	(*śmieci*)
	tonExecute															: TON;		
	tonNotExecute														: TON;	
	tonDelayAfterStart6s              									: TON;
	tonReadedCardFirstDelayBottleTransfer								: TON;
	tonReadedCardSecondDelayBottleTransfer								: TON;
	tonFourthFormatSensor												: TON;
	tonFourthFormatSensor2												: TON;	
	tonThirdFormsSensor													: TON;
	tonWaitUntilSecondFormPresent										: TON;
	tonLongDelayFirstDraging											: TON;
	tonLongDelayFirstDragingLidFeeder									: TON;	
	tonLongDelayFirstDragingLidSealer									: TON;	
	tonWeightBeforeGateDispSensor										: TON;
	tonBeforeGateSensorDelay											: TON;
	tonTransporterStopping												: TON;
	TimerCycleReseting													: TON;
	tonAfterScreweEmpty													: TON;
	tonCapCorrectCheckAfterScrewerFormSensor							: TON;
	fbbCapCorrectCheckAfterScrewerFormSensor							: FB_InputFilter_v2;
	tonDelayAfterReset													: TON;
	tonCycleLabelMachineFullSensor										: TON;
	tonCycleBadBottleConveyorFullSensor									: TON;
	tonCycleBadBottleConveyorFullSensor2								: TON;
	tofBadBottleConveyorStart											: TOF;
	tofbFormTransportersDispencerSlow									: TOF;
	tonbFormTransportersDispencerResetSpeed								: TON;
	tonQueBeforeScrewers												:TON;
	tonQueAfterScrewers													:TON;
	tonTimer4thFormBeforeCapSorter										:TON;
	tonQueAfterPlatin													:TON;
	tonQueBeforeDispencers												:TON;
	tonDelayedStartAfterDisp											:TON;
	
	i																	: UINT;
	nCheckCountR4														: UINT;
	iFormatOnWeightCounter												: UINT;
	cpc																	: INT;
	nccc																: INT;
	iBottleTransferCase													: INT;
	nCheckCountR1														: INT;
	iii																	: INT;
	iDispDragCase														: INT;
	iWeightCase															: INT;
	iScrewerDragCase													: INT;
	nw																	: INT;
	nw3																	: INT;
	nw2																	: INT;
	nw4																	: INT;
	nw5																	: INT;
	nw6																	: INT;
	nCounterFormsToLoad													: INT;
	nCounterForms														: INT;
	z																	: INT;
	iRobotPickCase														: INT;
	y																	: INT;
	nCounterCase7														: INT;
	nCounterCase8														: INT;
	nCounterCase10														: INT;
	nCounterCase14														: INT;
	nCounterCase11														: INT;
	nCounterCase12														: INT;
	cch																	: INT;
	cchc																: INT;	
	jw1																	: INT;
	jw2																	: INT;
	iw3																	: INT;
	jw3																	: INT;
	iw4																	: INT;
	jw4																	: INT;
	iw5																	: INT;
	jw5																	: INT;
	iw6																	: INT;
	jw6																	: INT;
	ic1																	: INT;
	iCOunterTest10														: INT;
	iWeightOnFormCase													: INT;
	nCountTest2															: INT;
	nCountTest3															: INT;
	iGateDispCase														: INT;
	counterchecked														: INT;
	nCounterCase9														: INT;
	nCounterCase13														: INT;
	nCounterCase15														: INT;
	ibRobotPackageState1NOK												: INT;
	iBeforeDispencerCounter												: INT;
	bRobotCycleRFIDReadedOne											: BOOL;
	bRobotCycleRFIDReadedTwo											: BOOL;
	bBadBottleConveyorStartTrigger										: BOOL;
	bBadBottleConveyorStartTriggerDelay									: BOOL;	
	bRobotGateStayOpen													: BOOL;
	bRobotPackageState1OK												: BOOL;
	bRobotPackageState1NOK												: BOOL;
	bRobotPackageState2OK												: BOOL;
	bRobotPackageState2NOK												: BOOL;
	bRobotPackageState1Rotate											: BOOL;
	bRobotPackageState2Rotate											: BOOL;
	iChangeModeStep: INT;
	bCatchersReady2														: BOOL;
	bDispencer2CatchedOrNoBottle										: BOOL;
	bDispencer1CatchedOrNoBottle										: BOOL;
	bDispencer3CatchedOrNoBottle										: BOOL;
	bDispencer4CatchedOrNoBottle										: BOOL;
	bCounterDisabled													: BOOL;
	bRobotPackageState1Empty											: BOOL;
	bRobotPackageState2Empty											: BOOL;
	//ctdCounterFormOnRobot												: CTD;
	iResetAfterErrorOrEstop: INT;
	iBeforeDispencer2PhaseCounter: INT;
	bBottleFeederHommed: BOOL;
	iFormatOnWeight2PhaseCounter: UINT;
	tonCheckFourthFormNotPresent: TON;
	tonFourthFormat2PhaseSensor: TON;
	tonCheckFormSensorBetweenDispencer: TON;
	ftfbIbWeightFirstForm2PhaseSensor: F_TRIG;
	iPhaseChangingStep: INT;
	tonPhaseChangingCase110Delay: TON;
	tonPhaseChangingCase200Delay: TON;	
	tonPhaseChangingCase210Delay: TON;
	iTestDrag: INT;
	brtLongDelayFirstDraging: BOOL;
	bFirstDragingLidFeederAfterRestart1: BOOL;	
	bFirstDragingLidFeederAfterRestart2: BOOL;	
	bFirstDragingLidSealerAfterRestart1: BOOL;	
	bFirstDragingLidSealerAfterRestart2: BOOL;		
	tonSecondForm2PhaseSensor: TON;
	bPhaseChangingGatePermission: BOOL;
	brtLongDelayFirstDragingDone: BOOL;
	brtLongDelayFirstDragingLidFeederDone: BOOL;	
	bDelayAfterStartFullRegister: BOOL;
	tonSecondForm2PhaseSensorRepair: TON;
	tonGripperScrewerDragMiddleSensor: TON;
	tonDispencersDragLeftMiddleSensor: TON;
	tonDispencersDragRightMiddleSensor: TON;
	tonDelayAfterBottleFeederDoorOpen: TON;
	tonCheckFormBeforeDispencersGate: TON;
	fbIbFourthFormCheckFormSensor: FB_InputFilter_v2;
	fbIbTwoPhasesFormSensorBetweenDispencers: FB_InputFilter_v2;
	fbIbSecondFormCheckFormSensor: FB_InputFilter_v2;
	tofbDosingTwoPhases:TOF;
	tonNotLongDelayAfterStart: TON;
	nVarModuloSimulation: INT;
	tonNotReadedCardFirstDelayBottleTransfer: TON;
	tonNotReadedCardSecondDelayBottleTransfer: TON;
	fbIbBottleTransferFormAfterSensor: FB_InputFilter_v2;
	rttonNotReadedCardFirstDelayBottleTransfer: R_TRIG;
	rttonNotReadedCardSecondDelayBottleTransfer: R_TRIG;
	iCounterRepairNotReadedFirst: INT;
	iCounterRepairNotReadedSecond: INT;
	rtbRobotPackageState1NOK: R_TRIG;
	rtbRobotPackageState2NOK: R_TRIG;
	ibRobotPackageState2NOK: INT;
	fbIbGripperScrewersThirdFormCheckFormSensor:FB_InputFilter;
	fbIbGripperScrewersBeforeThirdFormCheckFormSensor:FB_InputFilter;
	tofFormsDragingPneumaticStationDraged	:	TOF;
	toffbDispencersDragLeftStationbCycleDone: TOF;
	tonWeight14CycleDoneAndCase: TON;
	tonWeight56CycleDoneAndCase: TON;	
	iFormTransportersScrewerResetSpeedPulse: INT;

	
	(*CapSorter*)
	tonCapSorterDragMiddleSensor			:TON;
	tonIbCapSorterAfterFormSensor			:TON;
	tonIbCapSorterAfterFormSensor3			:TON;	
	brtCapSorterLongDelayFirstDraging		:BOOL;
	bCapSorterDragIfNot4PucksAnd5s			:BOOL;	
	tonCapSorterDragIfNot4PucksAnd5s		:TON;
	tonCapSorterFourthFormatSensorAnRegister:TON;
	tonIbCapSorterFirstFormCheckFormSensor	:TON;
	tonCapSorterFourthFormatSensor			:TON;
	tonCapSorterFourthFormatSensorStarting	:TON;	
	tonbFormTransportersAfterCapSorterCmdStart:TON;
	rttonCapSorterFourthFormatSensorCounter	:R_TRIG;
	tonCapSorterDragFormCounter4			:TON;
	tonCapSorterDragFormCounter4b			:TON;	
	itonCapSorterDragFormCounter4			:INT;
	itonCapSorterDragFormCounter4b			:INT;
	tonStoppingCapSorter					:TON;
	tonCapSorterDelay						:TON;
	tonCapSorterDelay2						:TON;
	iCapSorterCase							:INT;
	bDelayAfterStartCapSorterFullRegister	:BOOL;
	(*inne*)
	//Vasyl 30.05 
	tonPucksInserterPushTableOff			:TON;

	(*Szalaban przed waga*)
	iWeightGateBeforeCASE					: INT;													
	
	(*Zatrzymywanie transportera*)
	tonCapSorterCycleTime					: TON;
	fttonCapSorterCycleTime					: F_TRIG;
	AtCapSorterCycleTime					: ARRAY [1..100] OF TIME;
	bCapSorterCycleTest						: BOOL ;
	tonCapSorterPackageState1bCapSorterPutted: TON;
	tCapSorterCycleTestTime					: TIME;
	
	(*Wbijak butelek*)
	bBottlePusherBottleBeforeSensor			: BOOL;
	tonBottlePusherBottleBeforeSensor		: TON;
	
	
	(*AutoStart ADS*)
	tonBottleSorterAutoStart 				: TON;
	tonCapSorterAutoStart					: TON;
	iBottleSorterAutoStart 					: INT;	
	iCapSorterAutoStart						: INT;
	bCapSorterBottleSorterAutoStart 		: BOOL;	
	tonbCapSorterBottleSorterAutoStart 		: TON;
	
	(*Dodatkowe sprawdzanie butelki*)

	rtIbCapCorrectCheckFormSensor			: R_TRIG;
	
	(*Inne*)
	
	iAbortingTest: INT;
	iChooseRecipe: INT;

	toniWeight14GateBeforeCASE: TON;
	toniWeight14GateBeforeCASE2: TON;
	fbIbWeight14Gate4FormBeforeSensor: FB_InputFilter_v2;
	tonbGateBeforeWeight14Run: TON;
	toniWeight56GateBeforeCASE: TON;
	toniWeight56GateBeforeCASE2: TON;
	fbIbWeight56Gate6FormBeforeSensor: FB_InputFilter_v2;
	tonbGateBeforeWeight56Run: TON;
	
	ics: INT;
	ttonCapSorterCycleTimeET: TIME;
	bCapSorterError: BOOL;
	tonbCapSorterError: TON;
	tonbCapSorterOrCapSorterDragError: TON;	
	fbDrand: DRAND;
	diRandom :DINT;
	iTestResetCommandsStopped: INT;
	tonCapSorterHomingAndDone: TON;
	tonBottleSorterHomingAndDone: TON;
	irtResetAfterStart: INT;
	ibDelayAfterStartCapSorterFullRegister: INT;
	toniHomingCase20: TON;
	iTestiHomingCase: INT;

	bStopping1Weight: BOOL;
	bStoppingWeight1: BOOL;
	bStoppingWeight2: BOOL;
	bStoppingWeight3: BOOL;
	bStoppingWeight4: BOOL;
	tonStoppingBottleTransfer1: TON;
	
	tonbFirstCycle: TON;
	iTestW: INT;
	
	(*Wydmuch przed zakręcarkami*)
	fbIbBlowBeforeGripperScrewerSensor	:	FB_InputFilter_v2;
	fbIbBlowBeforeGripperScrewerSensor2	:	FB_InputFilter_v2;
	
	(*Licz form. przed doz*)
	rtIbFourthFormCheckFormSensor:	R_TRIG;
	tonIbFourthFormCheckFormSensor: TON;
	tonFormsDragingFormCounter4	: TON;
	tonFormsDragingFormCounter4b: TON;	
	itonFormsDragingFormCounter4: INT;	
	itonFormsDragingFormCounter4b: INT;
	
	(*Szlaban przed zakrecarkami*)
	fbIbGateBeforeGripperScrewerSensor						: FB_InputFilter;
	fb2IbGateBeforeGripperScrewerSensor						: FB_InputFilter;	
	ftfbIbGateBeforeGripperScrewerSensor					: F_TRIG;
	bGateBeforeGripperScrewer								: BOOL;
	tonbGateBeforeGripperScrewer							: TON;
	
	(*Lid Feeder Drag*)
	iLidFeederDragCase										: INT;	
	tofbLidFeederDragingStationPrepareRun					: TOF;
	tonLidFeederFirstFormSensorBeforeDrag					:TON;
	iLidFeederDragStoppingCount								: INT;
	bLidFeederDragDelayAfterStartFullRegister				: BOOL;	
	tonLidFeederDragSecondFormSensor						: TON;
	fbIbLidFeederAfterSensor								: FB_InputFilter_v2;
	fbIbLidFeederAfterSensorLonger							: FB_InputFilter_v2;
	tonAfterLidFeederEmpty									: TON;
	tonLidFeederThirdFormsSensor							: TON;
	fbIbLidFeederThirdFormCheckFormSensor					: FB_InputFilter_v2;
	bLidFeederReady											: BOOL;
	fb2IbLidFeederThirdFormSensor							: FB_InputFilter_v2;
	tonStartLidFeederDelay									: TON;
	iLidFeederCase											: INT;
	tonfbLidFeederDragStationNotbCycleDone					: TON;		
	(*Lid Putted Check*)
	fbIbLidPuttedCheck1Sensor								: FB_InputFilter_v2;
	fbIbLidPuttedCheck2Sensor								: FB_InputFilter_v2;
	
	
	(*Lid Sealer Drag*)
	iLidSealerDragCase										: INT;
	tofbLidSealerDragingStationPrepareRun					: TOF;
	iLidSealerDragStoppingCount								: INT;
	bLidSealerDragDelayAfterStartFullRegister				: BOOL;	
	tonLidSealerDragSecondFormSensor						: TON;
	fbIbLidSealerAfterSensor								: FB_InputFilter_v2;
	fbIbLidSealerAfterSensor2								: FB_InputFilter_v2;
	tonLidSealerThirdFormsSensor							: TON;
	tonLidSealerFirstFormsSensor								: TON;
	fbIbLidSealerThirdFormCheckFormSensor					: FB_InputFilter_v2;
	bLidSealerReady											: BOOL;
	fb2IbLidSealerSecondFormSensor							: FB_InputFilter_v2;
	fbNotIbLidSealerSecondFormSensor							: FB_InputFilter_v2;	
	tonStartLidSealerDelay									: TON;
	iLidSealerCase											: INT;	
	tonbFormTransportersScrewerCmdStart						: TON;
	tonfbLidSealerDragStationNotbCycleDone					: TON;		
	rttonLidSealerSecondFormatSensorCounter					: R_TRIG;
	tonLidSealerSecondFormatSensor							: TON;
	tonLidSelaerDragIfNot2PucksAnd5s						: TON;
	bLidSelaerDragIfNot2PucksAnd5s							: BOOL;
	(*Transfer na wagę*)
	udiBottleTransferWeightIntervalCount: UDINT;
	bBottleTransferDoWeight: BOOL;
	
	(*Inne*)
	iGateBeforeGripperScrewerCase: INT;
	toniGateBeforeGripperScrewerCase1: TON;
	tonBadBottleConveyorStop: Ton;
	
	
	toWeightRealeseByLidFeeder: TON;

	tonbFormTransportersScrewerStop: TON;
	tofFormTransportersScrewerSlowSpeed: TOF;
	iFirstDragingLidFeederAfterRestart2Count: INT;
	iFirstDragingLidSealerAfterRestart2Count: INT;	
	tonP13_BottleTransferfbBottleTransfereRunningStateeRejecting: TON;
	nUnderCorrectCapPackageStateLastnCardNumber: ULINT;
	nCapCorrectCheckCameraNOK: INT;
	rtP11_CapCorrectCheckfbCapCorrectCheckCamerabCycleDone: R_TRIG;
	nCapCorrectCheckCameraOK: INT;
	tonDragAE1: TON;
	
	(*Spowalniacz*)
	tonCapPuttedFormsCheck						:	TON;
	tonThirdFormCheckFormSensor					:	TON;
	
	(*SignalFormCounting*)
	fbIbCapSorterGateScrewerSensor: FB_InputFilter_v2;
	fbIbCapSorterGateWeightSensor: FB_InputFilter_v2;
	fbIbCapCorrectCheckFormSensor: FB_InputFilter_v2;

	(*PucksInserter*)
	bPucksInserterHommed: BOOL;

	(*inne*)
	iSetNumbersOfFormsBetweenWeightAndScrewers: INT;
	tofCapCorrectCheckAfterScrewerFormSensor: TOF;

	itonWeightPackageState1BnNoCardNumber: INT;
	itonWeightPackageState2BnNoCardNumber: INT;
	itonWeightPackageState3BnNoCardNumber: INT;
	itonWeightPackageState4BnNoCardNumber: INT;
	tonBreakpoint: TON;
	bBreakpoint: BOOL;
	tontonDelayAfterStart: TON;
	tonDelayForGatePI: TON;
	tonIbPucksInserterFormGateBeforeSensor: TON;

	(*ROPP*)
	fbIbROPPThirdFormSensor					:FB_InputFilter_v2; 
	rtfbIbROPPThirdFormSensor				:R_TRIG;
	rtfbIbROPPThirdFormSensor2				:R_TRIG;	
	ftfbIbROPPThirdFormSensor				:F_TRIG;
	tonROPPThirdFormSensor					:TON;
	tonROPPThirdFormSensor2					:TON;
	tonROPPAfterFormSensor					:TON;
	fbIbROPPAfterFormSensor 				:FB_InputFilter_v2; 
	fbIbROPPAfterFormSensor2 				:FB_InputFilter_v2; 
	fbIbROPPAfter3FormSensor 				:FB_InputFilter_v2; 
	ftIbROPPAfterFormSensor 				:F_TRIG; 
	iROPPAfterFormCounter					:INT;
	iROPPBeforeFormCounter					:INT;
	iTestRop1:INT;
	fbIbROPPSevenFormSensor					:FB_InputFilter_v2; 
	fbIbROPPSevenFormSensor2				:FB_InputFilter_v2; 
	rtfbIbROPPSevenFormSensor2				:R_TRIG;
	ftfbIbROPPSevenFormSensor2				:F_TRIG;
	ftbReadedCardBeforeROPP					:F_TRIG;
	tonbReadedCardBeforeROPP				:TON;
	fbbReadedCardAfterROPP					:FB_InputFilter_v2; 
	rtfbbReadedCardAfterROPP				:R_TRIG;
	ftfbbReadedCardAfterROPP				:F_TRIG;	
	rpc,rpc1,rcc,rcc1						:INT;
	bROPPReady								:BOOL;
	bROPPDelayAfterStartFullRegister		:BOOL;
	tonROPPStartCappingDelay				:TON;
	tofbROPPCappingRunEngine				:TOF;
	iROPPCappingCase						:INT;
	rtiROPPAfterFormCounter0				:R_TRIG;
	bDragTest								:BOOL;
	fbROPPIbCapSorterBeforeFourthFormCheckFormSensor:FB_InputFilter_v2; 
	iTestBot :INT;
	bTestBot:BOOL;
	BtESTbOT1:BOOL;
	iFormBeforeScrewers:INT;
	iFormBeforeROPP:INT;
	//bBlowBeforeGripperScrewer:BOOL;
	//tonbBlowBeforeGripperScrewer:TON;
	//tonQbBlowBeforeGripperScrewer:TON;
	tonIbROPPBeforeSevenFormSensor:TON;
	tpfbIbBlowBeforeGripperScrewerSensor:TP;
	iCaseSingleRealeseIfNoCapFromScrewersPulse:INT;
	tonSingleRealeseIfNoCapFromScrewers1:TON;
	tonSingleRealeseIfNoCapFromScrewers2:TON;	
	bSingleRealeseIfNoCapFromScrewersDragBlock: BOOL;
	rtSingleRealeseIfNoCapFromScrewers1:R_TRIG;
	rtSingleRealeseIfNoCapFromScrewers2:R_TRIG;
	tonBlowBeforeGripperScrewerSensor: TON;
	fbIbPucksInserterFormGateAfterSensor :FB_InputFilter_v2;
	fbIbPucksInserterPushTablesSensor :FB_InputFilter_v2;
	tofIbCapCorrectCheckFormSensor:TOF;
	bCapCorrectCheckBottleSensorLast:BOOL;
	iCapCorrectCheckBottleSensorLast:INT;
	bCapSorterDragIfNot4PucksAnd5sRepair:BOOL;
	fbTransporterQueues: FB_InputFilter_V2;
	fbIbDispencerAfterCheckFormSensor: FB_InputFilter_v2;
	fbIbDispencer12NoColisionWhenDosingSensor: FB_InputFilter_v2;
	fbIbDispencer34NoColisionWhenDosingSensor: FB_InputFilter_v2;	
	fbIbCapSorterFourthFormCheckFormSensor: FB_InputFilter_v2;
	rttofIbCapCorrectCheckFormSensor: R_TRIG;
	ibFormsDragingRightRun:INT;
	ibFormsDragingLeftRun:INT;	
	ftbFormsDragingRightRun:F_TRIG;
	ftbFormsDragingLeftRun:F_TRIG;
	rtbFormsDragingLeftRun	:R_trig;
	rtbFormsDragingRightRun	:R_trig;
	
	(*Szlaban na trans odbviorczym*)
	fbIbExitConveyorGateAfterSensor		:FB_InputFilter_v2;
	fbIbExitConveyorGateAfterSensor2	:FB_InputFilter_v2;	
	fbIbExitConveyorGateAfterSensor3	:FB_InputFilter_v2;	
	tonbExitConveyorGateRun				:TON;
	bExitConveyorGateRunTemp			:BOOL;
	(*Koniec Szlaban na trans odbviorczym*)
	bSafetyTest							:BOOL;
	
	lrGripperScrewerStoperPosition		:LREAL;
	tpGripperScrewerStoperTimerOn		:TP;	// timer do generowania impulsu
	fbGripperScrewerStoperSensorDelay	:FB_InputFilter;	// filtr do generowania sygnału 
	tofQbGripperScrewerStoperActuator	:TOF;	
	rtQbGripperScrewerStoperActuator	:R_TRIG;
	fbQbGripperScrewerGateBeforeActuator:FB_InputFilter_v2;	
	rtfbQbGripperScrewerGateBeforeActuator:R_TRIG;	
	bGripperScrewerStoper2ReadyToDrag 	:BOOL;
	tonQbGripperScrewerGateBeforeActuator:TON;
	itestdpvs			:INT;
	itestdpvs2			:INT;
	itestdpvs3			:INT;	
	bEXPACK	:BOOL:=FALSE;
	tofWeight6FormSensor	:TOF;
	tofbacktodrag			:TOF;
	tofQueAfterPlatinForDisp	:TOf;
	tonQueBeforePlatins	:TON;
	bGripperScrewerAcceleratorActuatorTemp: BOOL;
	tonDelayLid1Putting	:TON;
	tonDelayLid2Putting	:TON;
	
	
	//P13_BottleTransferAfterDrag
	tonBottleTransferAfterDrag	: TON;
	fbIbBottleTransferAfterDragAfterSensor : FB_InputFilter_v2;
	fbIbBottleTransferAfterDragSecondFormSensor	 : FB_InputFilter_v2;
	rtfbIbBottleTransferAfterDragSecondFormSensor : R_TRIG;
	rtfbIbBottleTransferAfterDragSecondFormSensorCounter : INT;
	tonrtfbIbBottleTransferAfterDragSecondFormSensorCounter: TON;
	// Konie cP13_BottleTransferAfterDrag
	
	(*Wick Feeder*)
	iWickFeederDragCase										: INT;	
	tofbWickFeederDragingStationPrepareRun					: TOF;
	tonWickFeederFirstFormSensorBeforeDrag					:TON;
	iWickFeederDragStoppingCount							: INT;
	bWickFeederDragDelayAfterStartFullRegister				: BOOL;	
	tonWickFeederDragSecondFormSensor						: TON;
	fbIbWickFeederAfterSensor								: FB_InputFilter_v2;
	fbIbWickFeederAfterSensorLonger							: FB_InputFilter_v2;
	tonAfterWickFeederEmpty									: TON;
	tonWickFeederThirdFormsSensor							: TON;
	fbIbWickFeederThirdFormCheckFormSensor					: FB_InputFilter_v2;
	bWickFeederReady										: BOOL;
	fb2IbWickFeederThirdFormSensor							: FB_InputFilter_v2;
	tonStartWickFeederDelay									: TON;
	iWickFeederCase											: INT;
	tonfbWickFeederDragStationNotbCycleDone					: TON;		
	tonDelayWick1Putting									: TON;
	tonDelayWick2Putting									: TON;
	bFirstDragingWickFeederAfterRestart1					: BOOL;	
	bFirstDragingWickFeederAfterRestart2					: BOOL;	
	iFirstDragingWickFeederAfterRestart2Count				: INT;
	(*Koniec Wick Feeder Drag*)
	
		//CapPusher
	iCapPusherGateCase			: INT;
	fbIbCapPusherFormSensor 	: FB_InputFilter_v2;
	fbIbCapPusherFormSensor2 	: FB_InputFilter_v2;	
	rtfbIbCapPusherFormSensor2 	: R_TRIG;		
	iCapPusherCase				: INT;	
	ftbReadedCard2				: F_TRIG;
	tonCapPusherDelay			: TON;
	tonCapPusherFormNotPresent	: TON;
	itonCapPusherFormNotPresent	: INT;
	//Koniec CapPusher
	
END_VAR

VIS.bServiceMode;
fbPMLModeManager.eModeStatus;
fbPMLAuto.ePMLState;
fbPMLManual.ePMLState;

ACT_CycleStarting();
ACT_CycleLogicInIdle();
ACT_Signals();
ACT_SignalsROPP();
ACT_SignalsLidFeeder();
ACT_ResetAfterStart();
ACT_Mode();
ACT_HomingCanceled();
ACT_CycleReset();
//ACT_PMLErrors();
ACT_HandlingCommands();
ACT_PMLModeManager();
ACT_PMLStates();
ACT_PMLResetCommands();
ACT_AntyError();
ACT_ResetAfterError();
ACT_Statistics();
ACT_SafetyFirstResetDelay();

ACTION ACT_Aborted:

ACT_ResetCommands();
END_ACTION

ACTION ACT_Aborting:
//Reset komunikatów z Visualization
P00_Visualization.aResetDialog();

//Sprawdzam czy każda stacja przeszła Aborting

//CapUnboxer
//bCapUnboxerAbortingState := GvlCommunication.stCapUnboxerRead.ePackMLAutoState <>  Tc3_PackML.E_PMLState.ePMLState_ABORTING OR NOT GvlCommunication.stCapUnboxerRead.bEnable OR bCapUnboxerDisabled;

//JarUnboxer
//bJarUnboxerAbortingState := GvlCommunication.stJarUnboxerRead.ePackMLAutoState <>  Tc3_PackML.E_PMLState.ePMLState_ABORTING OR NOT GvlCommunication.stJarUnboxerRead.bEnable OR bJarUnboxerDisabled;

//eDisabled := 0,eAborted := 1, eAborting := 2,	eError := 3, 
(*Aborted lub Disabled*)
IF 	
	P01_BottleFeeder.fbBottleFeeder.eState<=2 AND
	P01_BottleFeeder.fbTurnTable.eState<=2 AND
	P01_PucksInserter.fbPucksInserter.eState<=2 AND
	P01_PucksInserter.fbTurnTable.eState<=2 AND		
	(
	gvlCommunication.stBottleSorterRead.ePackMLAutoState <> Tc3_PackML.E_PMLState.ePMLState_ABORTING OR 
	NOT gvlCommunication.stBottleSorterRead.bEnable OR bBottleSorterDisable
	) AND
	P02_Dispencers.fbDispencersDragRightStation.eState<=2 AND
	P02_Dispencers.fbDispencersDragLeftStation.eState<=2 AND
    P02_Dispencers.fbDispencer1.eState <= 2 AND
    P02_Dispencers.fbDispencer2.eState <= 2 AND
    P02_Dispencers.fbDispencer3.eState <= 2 AND
    P02_Dispencers.fbDispencer4.eState <= 2 AND
    P02_Dispencers.fbDispencersCatch1Station.eState <= 2 AND
    P02_Dispencers.fbDispencersCatch2Station.eState <= 2 AND
    P02_Dispencers.fbDispencersCatch3Station.eState <= 2 AND
    P02_Dispencers.fbDispencersCatch4Station.eState <= 2 AND
    P05_Weight.fbWeight1.eState <= 2 AND
    P05_Weight.fbWeight2.eState <= 2 AND
    P05_Weight.fbWeight3.eState <= 2 AND
    P05_Weight.fbWeight4.eState <= 2 AND	
    P05_Weight.fbWeight5.eState <= 2 AND
    P05_Weight.fbWeight6.eState <= 2 AND ((	
	P05_Weight.fbWeightStation.eState <= 2 AND NOT VIS.bDosingTwoPhasesShow) OR ( P05_Weight.fbWeightStation2Phase.eState <= 2 AND  VIS.bDosingTwoPhasesShow)) AND
	
	P06_WickFeeder.fbWickFeederSt.eState <=2 AND
	P06_WickFeeder.fbWickFeederDragStation.eState <= 2 AND
	
	P06_LidFeeder.fbLidFeeder.eState <= 2 AND
	P06_LidFeeder.fbLidFeeder2.eState <= 2 AND
	P06_LidFeeder.fbLidFeederDragStation.eState <= 2 AND
	P06_LidPuttedCheck.fbLidPuttedCheck.eState <= 2 AND
	P06_LidSealer.fbLidSealer.eState <= 2 AND 
	P06_LidSealer.fbLidSealer2.eState <= 2 AND
	P06_LidSealer.fbLidSealerDragStation.eState <= 2 AND 

	P07_ROPP.fbROPPSlower.eState	<= 2 AND
	P07_ROPP.fbROPPFeeder.eState	<= 2 AND
	P07_ROPP.fbROPPDrag.eState		<= 2 AND
	P07_ROPP.fbROPPCapping.eState	<= 2 AND
	
	P08_CapSorter.fbCapSorterDragStation.eState <= 2 AND
	P08_CapFeeder.fbCapFeeder.eState <= 2 AND	
	(
	gvlCommunication.stCapSorterRead.ePackMLAutoState <> Tc3_PackML.E_PMLState.ePMLState_ABORTING OR 
	NOT gvlCommunication.stCapSorterRead.bEnable OR bCapSorterDisable
	) AND
	P09_CapPuttedCheck.fbCapPuttedCheck.eState <= 2 AND
	P10_GripperScrewer.fb2GripperScrewer1.eState <=2 AND
	P10_GripperScrewer.fb2GripperScrewer2.eState <=2 AND	
	P10_GripperScrewer.fbGripperScrewersDragStation.eState <=2 AND
	P10_GripperScrewer.fbGripperScrewer1CatchStation.eState <=2 AND
	P10_GripperScrewer.fbGripperScrewer2CatchStation.eState <=2 AND 
	P11_CapCorrectCheck.fbCapCorrectCheck.eState <=2 AND
	P13_BottleTransfer.fbBottleTransfer.eState <=2 AND
	P14_BadBottleConyevor.fbBadBottleConveyor.eState <=2 AND
	P15_FormTransporters.fbFormTransporterDispencer.eState <=2 AND
	P15_FormTransporters.fbFormTransporterScrewer.eState <=2 AND	
	P15_FormTransporters.fbFormTransporterBeforeScrewer.eState <=2 		
    THEN
  	iAbortingTest	:=	iAbortingTest	+	1;
		
	   fbPMLAuto.StateComplete					:= TRUE; 
	   fbPMLManual.StateComplete				:= TRUE;
	  
	   ACT_ResetCommands();
   
END_IF
END_ACTION

ACTION ACT_AntyError:

END_ACTION

ACTION ACT_CapSorterBottleSorterAutoStart:
(*
Nazwa:			ACT_CapSorterBottleSorterAutoStart
Opis:			Ponowne uruchominie, jeżeli sie nie uruchmią sortery po ADSie
Wersja:			v0.1
Data:			2024-07-01
Autor:			DP
Urzadzenia:		
Konfiguracja:	
Info:
- Sprawdzanie po czasie czy sortery się uruchomiły
*)
tonBottleSorterAutoStart (IN:=	fbPMLAuto.ePMLState = Tc3_PackML.E_PMLState.ePMLState_EXECUTE AND NOT (stBottleSorterRead.ePackMLAutoState = Tc3_PackML.E_PMLState.ePMLState_EXECUTE) AND stBottleSorterRead.bEnable AND NOT bBottleSorterDisable AND 
								NOT bCapSorterBottleSorterAutoStart
						, PT:=T#10S);
IF 	tonBottleSorterAutoStart.Q THEN
	iBottleSorterAutoStart	:=	iBottleSorterAutoStart	+	1;
END_IF

tonCapSorterAutoStart (IN:= fbPMLAuto.ePMLState = Tc3_PackML.E_PMLState.ePMLState_EXECUTE AND NOT (stCapSorterRead.ePackMLAutoState = Tc3_PackML.E_PMLState.ePMLState_EXECUTE) AND stCapSorterRead.bEnable AND NOT bCapSorterDisable AND
							NOT bCapSorterBottleSorterAutoStart
						, PT:=T#10S);
IF 	tonCapSorterAutoStart.Q THEN
	iCapSorterAutoStart	:=	iCapSorterAutoStart	+	1;	
END_IF

IF tonBottleSorterAutoStart.Q OR tonCapSorterAutoStart.Q THEN
	bCapSorterBottleSorterAutoStart:= TRUE;
END_IF	

//Start na 3 sekundy
tonbCapSorterBottleSorterAutoStart	(IN:=	bCapSorterBottleSorterAutoStart, PT:= T#3S);
IF tonbCapSorterBottleSorterAutoStart.Q THEN
	bCapSorterBottleSorterAutoStart	:=	FALSE;
END_IF
END_ACTION

ACTION ACT_Clearing:
//eDisabled := 0,eAborted := 1, eAborting := 2,	eError := 3, 	
IF 
	
	P01_BottleFeeder.fbBottleFeeder.eState>2 OR P01_BottleFeeder.fbBottleFeeder.bEnable AND
	P01_BottleFeeder.fbTurnTable.eState>2 OR P01_BottleFeeder.fbTurnTable.bEnable AND
	P01_PucksInserter.fbPucksInserter.eState>2 OR P01_PucksInserter.fbPucksInserter.bEnable AND
	P01_PucksInserter.fbTurnTable.eState>2 OR P01_PucksInserter.fbTurnTable.bEnable AND	
	(
	(stBottleSorterRead.ePackMLAutoState <> Tc3_PackML.E_PMLState.ePMLState_ABORTING AND
	stBottleSorterRead.ePackMLAutoState <> Tc3_PackML.E_PMLState.ePMLState_ABORTED AND
	stBottleSorterRead.bEnable) OR NOT gvlCommunication.stBottleSorterRead.bEnable OR bBottleSorterDisable
	) AND
	P02_Dispencers.fbDispencersDragRightStation.eState >2 OR P02_Dispencers.fbDispencersDragRightStation.bEnable AND
	P02_Dispencers.fbDispencersDragLeftStation.eState >2 OR P02_Dispencers.fbDispencersDragLeftStation.bEnable AND
    P02_Dispencers.fbDispencer1.eState >2 OR P02_Dispencers.fbDispencer1.bEnable AND
    P02_Dispencers.fbDispencer2.eState >2 OR P02_Dispencers.fbDispencer2.bEnable AND
    P02_Dispencers.fbDispencer3.eState >2 OR P02_Dispencers.fbDispencer3.bEnable AND
    P02_Dispencers.fbDispencer4.eState >2 OR P02_Dispencers.fbDispencer4.bEnable AND
    P02_Dispencers.fbDispencersCatch1Station.eState >2 OR P02_Dispencers.fbDispencersCatch1Station.bEnable AND
    P02_Dispencers.fbDispencersCatch2Station.eState >2 OR P02_Dispencers.fbDispencersCatch2Station.bEnable AND
    P02_Dispencers.fbDispencersCatch3Station.eState >2 OR P02_Dispencers.fbDispencersCatch3Station.bEnable  AND
    P02_Dispencers.fbDispencersCatch4Station.eState >2 OR P02_Dispencers.fbDispencersCatch4Station.bEnable AND
    P05_Weight.fbWeight1.eState >2 OR P05_Weight.fbWeight1.bEnable AND
    P05_Weight.fbWeight2.eState >2 OR P05_Weight.fbWeight2.bEnable AND
    P05_Weight.fbWeight3.eState >2 OR P05_Weight.fbWeight3.bEnable AND
    P05_Weight.fbWeight4.eState >2 OR P05_Weight.fbWeight4.bEnable AND	
    P05_Weight.fbWeight5.eState >2 OR P05_Weight.fbWeight5.bEnable AND	
    P05_Weight.fbWeight6.eState >2 OR P05_Weight.fbWeight6.bEnable AND		
	P05_Weight.fbWeightStation.eState >2 OR P05_Weight.fbWeightStation.bEnable AND
	P05_Weight.fbWeightStation2Phase.eState >2 OR P05_Weight.fbWeightStation2Phase.bEnable AND
	P06_LidFeeder.fbLidFeeder.eState >2 OR P06_LidFeeder.fbLidFeeder.bEnable AND
	P06_LidFeeder.fbLidFeeder2.eState >2 OR P06_LidFeeder.fbLidFeeder2.bEnable AND
	P06_LidFeeder.fbLidFeederDragStation.eState >2 OR P06_LidFeeder.fbLidFeederDragStation.bEnable AND
	//P06_LidPuttedCheck.fbLidPuttedCheck.eState >2 OR P06_LidPuttedCheck.fbLidPuttedCheck.bEnable AND
	P06_LidSealer.fbLidSealer.eState >2 OR P06_LidSealer.fbLidSealer.bEnable AND 
	P06_LidSealer.fbLidSealer2.eState >2 OR P06_LidSealer.fbLidSealer2.bEnable AND
	P06_LidSealer.fbLidSealerDragStation.eState >2 OR P06_LidSealer.fbLidSealerDragStation.bEnable AND 

	P06_WickFeeder.fbWickFeederSt.eState >2 OR P06_WickFeeder.fbWickFeederSt.bEnable AND
	P06_WickFeeder.fbWickFeederDragStation.eState >2 OR P06_WickFeeder.fbWickFeederDragStation.bEnable AND

	P07_ROPP.fbROPPSlower.eState	>2 OR P07_ROPP.fbROPPSlower.bEnable AND
	P07_ROPP.fbROPPFeeder.eState	>2 OR P07_ROPP.fbROPPFeeder.bEnable AND
	P07_ROPP.fbROPPDrag.eState		>2 OR P07_ROPP.fbROPPDrag.bEnable AND
	P07_ROPP.fbROPPCapping.eState	>2 OR P07_ROPP.fbROPPCapping.bEnable AND

	P08_CapSorter.fbCapSorterDragStation.eState >2 OR P08_CapSorter.fbCapSorterDragStation.bEnable AND
	P08_CapFeeder.fbCapFeeder.eState >2 OR P08_CapFeeder.fbCapFeeder.bEnable AND	
	(
	(stCapSorterRead.ePackMLAutoState <> Tc3_PackML.E_PMLState.ePMLState_ABORTING AND
	stCapSorterRead.ePackMLAutoState <> Tc3_PackML.E_PMLState.ePMLState_ABORTED AND
	stCapSorterRead.bEnable OR bCapSorterDisable) OR NOT gvlCommunication.stCapSorterRead.bEnable
	) AND
	P09_CapPuttedCheck.fbCapPuttedCheck.eState >2 OR P09_CapPuttedCheck.fbCapPuttedCheck.bEnable AND
	P10_GripperScrewer.fb2GripperScrewer1.eState >2 OR P10_GripperScrewer.fb2GripperScrewer1.bEnable1 AND
	P10_GripperScrewer.fb2GripperScrewer2.eState >2 OR P10_GripperScrewer.fb2GripperScrewer2.bEnable1 AND	
	P10_GripperScrewer.fbGripperScrewersDragStation.eState >2 OR P10_GripperScrewer.fbGripperScrewersDragStation.bEnable AND
	P10_GripperScrewer.fbGripperScrewer1CatchStation.eState >2 OR P10_GripperScrewer.fbGripperScrewer1CatchStation.bEnable AND
	P10_GripperScrewer.fbGripperScrewer2CatchStation.eState >2 OR P10_GripperScrewer.fbGripperScrewer2CatchStation.bEnable AND 
	P11_CapCorrectCheck.fbCapCorrectCheck.eState >2 OR P11_CapCorrectCheck.fbCapCorrectCheck.bEnable AND
	P13_BottleTransfer.fbBottleTransfer.eState >2 OR P13_BottleTransfer.fbBottleTransfer.bEnable AND
	P14_BadBottleConyevor.fbBadBottleConveyor.eState >2 OR P14_BadBottleConyevor.fbBadBottleConveyor.bEnable AND
	P15_FormTransporters.fbFormTransporterDispencer.eState >2 OR P15_FormTransporters.fbFormTransporterDispencer.bEnable AND
	P15_FormTransporters.fbFormTransporterScrewer.eState >2 OR P15_FormTransporters.fbFormTransporterScrewer.bEnable AND	
	P15_FormTransporters.fbFormTransporterROPP.eState >2 OR P15_FormTransporters.fbFormTransporterROPP.bEnable AND	
	P15_FormTransporters.fbFormTransporterBeforeScrewer.eState >2 OR P15_FormTransporters.fbFormTransporterBeforeScrewer.bEnable		

    THEN
   
   fbPMLAuto.StateComplete						:= TRUE; 
   fbPMLManual.StateComplete					:= TRUE; 
   
END_IF
END_ACTION

ACTION ACT_CycleLogic:
	(*
TUTAJ
CAŁA 
LOGIKA
STEROWANIA
FBKAMI
*)


ACT_PhaseChanging(); //Procedura zmiany fazy (jednofazowe-dwufazowe)
aP00_SingleRealeseIfNoCapBeforeScrewers();
aP01_Gates();
aP01_GatesLidFeederBarrier();
aP01_Barriers();
aP01_BottleFeeder();
aP01_PucksInserter();
aP01_BottleSorter();
aP02_BottlePusher();
IF bDosingTwoPhases THEN
	aP02_Drag2Phase_GateAfter();	
	aP02_Dispencers2Phase();	
ELSE
	aP02_Drag1Phase_GateAfter();	
	aP02_Dispencers1Phase();
END_IF
//aP02_DragCheck();
aP05_WeightGateBefore();
aP05_Weight();
aP05_WeightBlock();
aP06_LidFeeder();
aP06_LidPuttedCheck();
aP06_LidSealer();
IF tofbDosingTwoPhases.Q OR VIS.bDosingTwoPhasesShow THEN
	aP06_LidSealerDrag2Phase();
ELSE
	aP06_LidSealerDrag();
END_IF
aP06_WickFeeder();
aP07_ROPP();
aP08_CapFeeder();
aP08_CapSorter();
aP09_CapPuttedCheck();
aP10_GripperScrewer();
aP10_GripperScrewerGate();
aP11_CapCorrectCheck();
aP13_BottleTransfer();
aP13_BottleTransferAfterDrag();
aP14_BadBottleConveyor();
aP15_FormTransporters();
aP16_LabelMachines();
END_ACTION

ACTION ACT_CycleLogicInIdle:
aP17_TurnTables();
aP02_DragCheck();
END_ACTION

ACTION ACT_CycleReset:
(*
Nazwa:			aCycleReset
Opis:			Restowanie cyklu
Wersja:			v0.1
Data:			2018-10-10
Autor:			
Urzadzenia:		
Konfiguracja:	
Info:
*)

(*Resetowanie cyklu , tylko gdy maszyna jest w gotowości *)
rtCycleReseting(CLK:=bCycleReseting, Q=>);
	
IF bCycleReseting THEN // Trwa 1 sek
	bLongDelayAfterStart		:=	FALSE;
	(*Resetowanie*)
	(*...*)
	(*****************KONIEC ZAPISYWANIE RFID*********************)
//Kasowanie tablicy RFID
	FOR i := 1 TO 100 DO //Dodane  bo KK
			eRFID[i] := eClearPackageState;
			
	END_FOR	


	VIS.bWeightCorrectionReset			:=	TRUE;
	iDispencersCase						:=	0;
	iWeightCase							:=	0;
	iDispDragCase						:=	0;
	
	VIS.bGateBeforeWeight14Run			:=	FALSE;
	VIS.bGateBeforeWeight56Run			:=	FALSE;
	iWeightGateBeforeCASE				:=	0;
	
	iScrewerDragCase					:=	0;
	iGripperScrewerCase					:=	0;
	iRobotPickCase						:=	0;
	iBottleTransferCase					:=	0;
	iWeightOnFormCase					:=	0;
	iGateDispCase						:=	0;
	bDragingFormsNotDone				:=	FALSE;
	bFormTransportersDispencerSlowSpeedPulse	:=  FALSE;
	bPhaseChangingGatePermission:=	FALSE;
	brtLongDelayFirstDragingDone	:=	FALSE;	
	IF bDosingTwoPhases THEN
		MAIN.aCycleRegister2Phase();
	ELSE
		MAIN.aCycleRegister1Phase();
	END_IF
	MAIN.aCycleRegisterROPP();
	
	
	MAIN.aStartingPoint();
	
	iLidSealerDragCase					:=	0;
	iLidSealerDragStoppingCount			:=	0;
	iWickFeederCase						:=	0;
	iWickFeederDragCase					:=	0;
	iWickFeederDragStoppingCount		:=0;	
	iLidFeederDragCase					:=	0;
	iLidFeederDragStoppingCount			:=	0;
	iLidFeederCase						:=	0;
	
	lrFormWeight1RFID					:=	0;
	lrFormWeight2RFID					:=	0;
	lrFormWeight3RFID					:=	0;
	lrFormWeight4RFID					:=	0;
	lrFormWeight5RFID					:=	0;
	lrFormWeight6RFID					:=	0;
	
ELSE 
	;
END_IF

IF rtCycleReseting.Q THEN
	GVL.bResetStates:=TRUE;
	ACT_ResetCommands();
		iCOunterTest10:=iCounterTest10+1;
	GVL.bDelay40sAfterReset:=TRUE;
	FOR i := 1 TO 17 DO 
		eBeforeROPPCapControlPackageState[i]	:=		eClearPackageState;
		eBeforeROPPPackageState[i]				:=		eClearPackageState;			
		eBeforeROPP2PackageState[i]				:=		eClearPackageState;		
		eUnderROPPPackageState[i]				:=		eClearPackageState;			
		eUnderROPPCorrectCapPackageState[i]		:=		eClearPackageState;
	END_FOR
END_IF

TimerCycleReseting();
TimerCycleReseting.IN:=bCycleReseting;
TimerCycleReseting.PT:=T#1S;

IF TimerCycleReseting.Q THEN
	bCycleReseting:=FALSE;
END_IF
END_ACTION

ACTION ACT_CycleStarting:

//Jezeli rozpoczęcie sie nie powiodło
IF bLongDelayAfterStart AND NOT tonLongDelayAfterStart.Q AND NOT (fbPMLAuto.ePMLState = Tc3_PackML.E_PMLState.ePMLState_EXECUTE) THEN
	bLongDelayAfterStart		:=	FALSE;
END_IF
END_ACTION

ACTION ACT_HandlingCommands:
rtStart															(CLK:= (IbCycleStartButton OR IbTurnTableCycleStartButton OR P07_ROPP.IbROPPCycleStartButton OR IbPucksInserterCycleStartButton OR
																		(stBottleSorterRead.bCycleStart AND NOT bBottleSorterDisable) OR
																		(stCapSorterRead.bCycleStart AND NOT bCapSorterDisable)) AND 
																		(*NOT bChangeover AND*) NOT bCIP AND bStationsAreReady);
	
tonStart														(IN:= (IbCycleStartButton OR IbTurnTableCycleStartButton OR P07_ROPP.IbROPPCycleStartButton OR IbPucksInserterCycleStartButton OR
																		(stBottleSorterRead.bCycleStart AND NOT bBottleSorterDisable) OR
																		(stCapSorterRead.bCycleStart AND NOT bCapSorterDisable)) AND 
																		(*NOT bChangeover AND*) NOT bCIP AND bStationsAreReady, PT:=T#2S);
															
ftStopCycle														(CLK:= 	NOT		IbCycleStopButton (*OR NOT IbTurnTableCycleStopButton OR NOT P07_ROPP.IbROPPCycleStopButton*) OR NOT IbPucksInserterCycleStopButton OR
																		(NOT	stBottleSorterRead.bCycleStop	AND NOT bBottleSorterDisable) OR 
																		(NOT	stCapSorterRead.bCycleStop		AND NOT bCapSorterDisable) 
																		
																		);
ftVisuReset														(CLK:= VIS.bResetErrorVisuCmd);
rtEstop															(CLK:= IbEmergencyStop);
rtResetAlarmTrigger												(CLK:= NOT IbCycleStopButton (*OR NOT IbTurnTableCycleStopButton*) (*OR NOT P07_ROPP.IbROPPCycleStopButton*) OR (IbCycleStartButton (*OR IbTurnTableCycleStartButton OR P07_ROPP.IbROPPCycleStartButton*)),		Q=>);
tonResetErrorVisuCmd											(IN:=nResetErrorVisuCmd>0,									PT:=T#500MS);


tpStopCycle.IN										:= ftStopCycle.Q OR tonConfectionEnding.Q;
tpStopCycle.PT										:= T#500MS;
tpStopCycle();

//Komenda Abort, brak safety
IF NOT IbEmergencyStop THEN
	fbPMLAuto.Abort									:= NOT IbEmergencyStop;
	fbPMLManual.Abort								:= NOT IbEmergencyStop;
END_IF

//Komenda Clear, safety - ok
IF IbEmergencyStop THEN
	fbPMLAuto.Clear									:= IbEmergencyStop; 
	fbPMLManual.Clear								:= IbEmergencyStop;
END_IF

//Komenda Stop
IF ftStopCycle.Q OR rtStopCycle.Q OR tonConfectionEnding.Q THEN
	fbPMLAuto.Stop									:= TRUE;  
	fbPMLManual.Stop								:= TRUE; 
END_IF

//Komenda Start
IF rtStart.Q THEN
	VIS.bCheckStart								 	:= TRUE; //Sprawdzanie czy zalogowany jest użytkownik na wizualizacji
END_IF
VIS.bAllowStart ;

//IF rtStart.Q THEN//THEN 					// Pozwolenie z wizualizacji 
IF VIS.bAllowStart  OR tonStart.Q THEN//THEN 					// Pozwolenie z wizualizacji 
	IF NOT VIS.bCapSorterEmptyingMode AND NOT VIS.bBottleSorterEmptyingMode THEN
		fbPMLAuto.Start									:= bStationsAreReady AND NOT bAtLeastOneOfTheStationsNeedHoming;
		fbPMLManual.Start								:= bStationsAreReady AND NOT bAtLeastOneOfTheStationsNeedHoming;
		//VIS.bAllowStart	:= FALSE;
		//VIS.bCheckStart	:= FALSE;
	END_IF
END_IF	

//Komenda Reset
IF ftVisuReset.Q  THEN
	fbPMLAuto.Reset									:= TRUE; 
	fbPMLManual.Reset								:= TRUE; 
END_IF

//Przejście Compliting
IF fbPMLAuto.ePMLState = Tc3_PackML.E_PMLState.ePMLState_COMPLETE THEN
	fbPMLAuto.Reset									:= TRUE; 
	fbPMLManual.Reset								:= TRUE; 
END_IF

IF fbPMLAuto.ePMLState <> Tc3_PackML.E_PMLState.ePMLState_STOPPING AND fbPMLAuto.ePMLState <> Tc3_PackML.E_PMLState.ePMLState_STOPPED THEN
	IF VIS.bErrorOccure THEN
		fbPMLAuto.Stop								:= TRUE;  
		fbPMLManual.Stop							:= TRUE; 
	END_IF
END_IF

//Tryb Serwisowy
IF VIS.bServiceMode AND fbPMLModeManager.eModeStatus = Tc3_PackML.E_PMLUnitMode.ePMLUnitMode_AUTOMATIC THEN
	//ACT_ResetCommands();
	
	//fbPMLModeManager.eModeCommand					:= Tc3_PackML.E_PMLUnitMode.ePMLUnitMode_MANUAL;
	//fbPMLModeManager.Execute						:= TRUE;
END_IF

//fbPMLModeManager();
IF NOT VIS.bServiceMode AND fbPMLModeManager.eModeStatus = Tc3_PackML.E_PMLUnitMode.ePMLUnitMode_MANUAL AND bStationsAreReadyOrError AND (stBottleSorterRead.ePackMLAutoState =  E_PMLState.ePMLState_IDLE OR NOT stBottleSorterRead.bEnable OR bBottleSorterDisable) AND (stCapSorterRead.ePackMLAutoState =  E_PMLState.ePMLState_IDLE OR NOT stCapSorterRead.bEnable OR bCapSorterDisable)  THEN
	//fbPMLModeManager.eModeCommand					:= Tc3_PackML.E_PMLUnitMode.ePMLUnitMode_AUTOMATIC;
	//fbPMLModeManager.Execute						:= TRUE;

	bManualMode								:= FALSE;
END_IF
ACT_PmlChangeMode();

//Wykrywanie blędu podczas ruchu
IF  (fbPMLAuto.ePMLState = Tc3_PackML.E_PMLState.ePMLState_EXECUTE OR fbPMLAuto.ePMLState = Tc3_PackML.E_PMLState.ePMLState_STOPPING) AND (VIS.bErrorOccure OR NOT IbEmergencyStop) THEN
	bResetAfterErrorOrEstop	:= TRUE;
	iResetAfterErrorOrEstop	:= iResetAfterErrorOrEstop	+	1;
END_IF


IF rtbRecipeLoading.Q THEN
	bRecipeChangePositioning 	:=	FALSE;
	bHomingCanceled				:=	FALSE;
END_IF
END_ACTION

ACTION ACT_HomingCanceled:


rtHomingIsOnAtLeastOneStation.CLK	:= 
									VIS.bBottleFeederHoming	OR	
									VIS.bPucksInserterHoming OR		
									stBottleSorterWrite.bHoming OR stBottleSorterRead.bHoming OR		
									VIS.bDispencersHoming OR     
									VIS.bFormsDragingRightHoming OR	
									VIS.bFormsDragingLeftHoming OR
									VIS.bWeightLiftHoming OR	
									VIS.bWickFeederHoming OR
									VIS.bWickFeederDragingHoming OR		
									VIS.bLidFeederHoming OR
									VIS.bLidFeederDragingHoming OR
									VIS.bLidPuttedCheckHoming OR
									VIS.bLidSealerHoming OR
									VIS.bLidSealerDragingHoming OR
									VIS_ROPP.bROPPFeederHoming OR	
									VIS_ROPP.bROPPDragHoming OR	
									VIS_ROPP.bROPPCappingHoming OR																																			
									VIS.bCapFeederHoming OR			
									VIS.bCapSorterDragHoming OR		
									stCapSorterWrite.bHoming OR stCapSorterRead.bHoming OR 			
									VIS.bCapPuttedCheckHoming OR		
									VIS.bGripperScrewerHoming OR		
									VIS.bBottleDragingStationHoming OR	
									VIS.bCapCorrectCheckHoming OR      
									VIS.bBottleTransferHoming  
									;
rtHomingIsOnAtLeastOneStation();
END_ACTION

ACTION ACT_HomingCycle:
//Obsługa HomingDialog
IF fbPMLAuto.ePMLState = Tc3_PackML.E_PMLState.ePMLState_RESETTING AND fbPMLModeManager.eModeStatus = Tc3_PackML.E_PMLUnitMode.ePMLUnitMode_AUTOMATIC THEN
	IF NOT bHomingCanceled AND bAtLeastOneOfTheStationsNeedHoming THEN
		bHomingDialog							:= TRUE;
	END_IF
END_IF



toniHomingCase20(IN:=iHomingCase=20,PT:=T#7S);
//Obsługa procedury bazowania
//Kiedy ? 1.Kiedy jakaś stacja nie zbazowana, 2.Po zmianie receptury
CASE iHomingCase OF

	0:
		IF bStationsAreReadyOrManual THEN
			IF bHoming THEN
				
				IF NOT bRecipeChangePositioning THEN
					bRecipeChangePositioning			:= VIS.bChooseRecipe;

				END_IF
				
				IF NOT bRecipeChangePositioning THEN
					IF fbPMLModeManager.eModeStatus = Tc3_PackML.E_PMLUnitMode.ePMLUnitMode_MANUAL THEN
						iHomingCase						:= 20;
					END_IF
					IF fbPMLModeManager.eModeStatus = Tc3_PackML.E_PMLUnitMode.ePMLUnitMode_AUTOMATIC THEN
						iHomingCase						:= 10;
					END_IF
				ELSE
					//stBottleSorterWrite.bHoming 		:= TRUE;
					//stCapSorterWrite.bHoming 			:= TRUE;
					iHomingCase							:= 5;
				END_IF
				
			END_IF	
		END_IF
		
	5: 

			VIS.bBottleFeederHoming			:= bBottleFeederEnable; 
			VIS.bPucksInserterHoming		:= bPucksInserterEnable; 			
			stBottleSorterWrite.bHoming 	:= NOT bBottleSorterDisable;
            VIS.bDispencersHoming           := bDispencer1Enable OR bDispencer2Enable OR bDispencer3Enable OR bDispencer4Enable;
			VIS.bFormsDragingRightHoming	:= GVL.bFormsDragingRightEnable;
			VIS.bFormsDragingLeftHoming		:= GVL.bFormsDragingLeftEnable;
			VIS.bWeightLiftHoming			:= GVL.bWeightLiftEnable;
			VIS.bCapFeederHoming			:= bCapFeederEnable;	
			VIS.bWickFeederHoming			:= bWickFeederEnable;
			VIS.bWickFeederDragingHoming	:= bWickFeederDragingStationEnable OR bWickFeederEnable;
			VIS.bLidFeederHoming			:= bLidFeederEnable (*OR bLidFeederDragingStationEnable*) ;
			VIS.bLidFeederDragingHoming		:= bLidFeederDragingStationEnable OR bLidFeederEnable;
			//VIS.bLidPuttedCheckHoming		:= bLidPuttedCheckEnable;
			VIS.bLidSealerHoming			:= bLidSealerEnable;
			VIS.bLidSealerDragingHoming		:= bLidSealerDragingStationEnable;
			VIS_CP.bCapPusherHoming 		:= bCapPusherHoming;
			VIS_CP.bCapPusherFeederHoming 	:= bCapPusherFeederHoming;
			VIS_ROPP.bROPPFeederHoming		:= bROPPFeederEnable;
			VIS_ROPP.bROPPDragHoming		:= bROPPDragEnable;
			VIS_ROPP.bROPPCappingHoming		:= bROPPCappingEnable;
			VIS.bCapSorterDragHoming		:= bCapSorterDragEnable;		
			stCapSorterWrite.bHoming 		:= NOT bCapSorterDisable;			
			VIS.bCapPuttedCheckHoming		:= bCapPuttedCheckEnable;
	        VIS.bGripperScrewerHoming		:= bGripperScrewer1Enable OR bGripperScrewer2Enable ;
			VIS.bBottleDragingStationHoming	:= bBottleDragingStationEnable; 
			VIS.bCapCorrectCheckHoming      := bCapCorrectCheckEnable;
			VIS.bBottleTransferHoming		:= bBottleTransferEnable;
			
			

			iHomingCase										:= 20; //10??
		
	10: //Wystawiam bazowanie gdy stacja nie zbazowana 

			VIS.bBottleFeederHoming		:= NOT P01_BottleFeeder.fbBottleFeeder.bHomingDone AND bBottleFeederEnable;	 //dodane Damian
			VIS.bPucksInserterHoming	:= NOT P01_PucksInserter.fbPucksInserter.bHomingDone AND bPucksInserterEnable;	 
			stBottleSorterWrite.bHoming := NOT bBottleSorterDisable;	
            VIS.bDispencersHoming         := (NOT P02_Dispencers.fbDispencer1.bHomingDone OR
                                             NOT P02_Dispencers.fbDispencer2.bHomingDone OR
                                             NOT P02_Dispencers.fbDispencer3.bHomingDone OR
                                             NOT P02_Dispencers.fbDispencer4.bHomingDone OR
                                             NOT P02_Dispencers.fbDispencersCatch1Station.bHomingDone OR
                                             NOT P02_Dispencers.fbDispencersCatch2Station.bHomingDone OR
                                             NOT P02_Dispencers.fbDispencersCatch3Station.bHomingDone OR
                                             NOT P02_Dispencers.fbDispencersCatch4Station.bHomingDone
                                                 ) AND
                                             (bDispencer1Enable OR bDispencer2Enable OR bDispencer3Enable OR bDispencer4Enable);
			//Bazpwanie przeciągania fomratek pod dozownikami
			
			VIS.bFormsDragingRightHoming		:= NOT P02_Dispencers.fbDispencersDragRightStation.bHomingDone AND bFormsDragingRightEnable;
			VIS.bFormsDragingLeftHoming			:= NOT P02_Dispencers.fbDispencersDragLeftStation.bHomingDone AND bFormsDragingLeftEnable;
			
			// Bazowanie wagi i szalek
			VIS.bWeightLiftHoming 			:=	(NOT P05_Weight.fbWeightStation.bHomingDone OR 
												NOT P05_Weight.fbWeightStation2Phase.bHomingDone) AND bWeightLiftEnable ;
			VIS.bWickFeederHoming			:=	(NOT P06_WickFeeder.fbWickFeederSt.bHomingDone  AND bWickFeederEnable);
			VIS.bWickFeederDragingHoming		:=	(NOT P06_WickFeeder.fbWickFeederDragStation.bHomingDone AND bWickFeederDragingStationEnable) OR (NOT P06_WickFeeder.fbWickFeederSt.bHomingDone  AND bWickFeederEnable); 

			VIS.bLidFeederHoming			:=	((NOT P06_LidFeeder.fbLidFeeder.bHomingDone OR NOT P06_LidFeeder.fbLidFeeder2.bHomingDone) AND bLidFeederEnable); //OR (NOT P06_LidFeeder.fbLidFeederDragStation.bHomingDone AND bLidFeederDragingStationEnable);
			VIS.bLidFeederDragingHoming		:=	(NOT P06_LidFeeder.fbLidFeederDragStation.bHomingDone AND bLidFeederDragingStationEnable) OR ((NOT P06_LidFeeder.fbLidFeeder.bHomingDone OR NOT P06_LidFeeder.fbLidFeeder2.bHomingDone) AND bLidFeederEnable); 
			//VIS.bLidPuttedCheckHoming		:=	(NOT P06_LidPuttedCheck.fbLidPuttedCheck.bHomingDone AND bLidPuttedCheckEnable);
			VIS.bLidSealerHoming			:=	((NOT P06_LidSealer.fbLidSealer.bHomingDone OR NOT P06_LidSealer.fbLidSealer2.bHomingDone) AND bLidSealerEnable);
			VIS.bLidSealerDragingHoming		:=	(NOT P06_LidSealer.fbLidSealerDragStation.bHomingDone AND bLidSealerDragingStationEnable);
			
			VIS.bWickFeederDragingHoming	:= NOT P06_WickFeeder.fbWickFeederDragStation.bHomingDone AND bWickFeederDragingStationEnable;
			VIS.bWickFeederHoming			:= NOT P06_WickFeeder.fbWickFeederSt.bHomingDone AND bWickFeederEnable;
			
			VIS_CP.bCapPusherHoming 		:= NOT P07_CapPusher.fbCapPusher.bHomingDone AND bCapPusherEnable;
			VIS_CP.bCapPusherFeederHoming 	:= NOT P07_CapPusher.fbCapPusherFeeder.bHomingDone AND bCapPusherEnable;
			

			VIS_ROPP.bROPPFeederHoming		:= NOT P07_ROPP.fbROPPFeeder.bHomingDone AND bROPPFeederEnable;
			VIS_ROPP.bROPPDragHoming		:= NOT P07_ROPP.fbROPPDrag.bHomingDone AND bROPPDragEnable;
			VIS_ROPP.bROPPCappingHoming		:= NOT P07_ROPP.fbROPPCapping.bHomingDone AND bROPPCappingEnable;

			//Bazpwanie podawania nakrętki
			VIS.bCapFeederHoming			:= NOT P08_CapFeeder.fbCapFeeder.bHomingDone AND bCapFeederEnable;									
			VIS.bCapSorterDragHoming		:= NOT P08_CapSorter.fbCapSorterDragStation.bHomingDone AND bCapSorterDragEnable;	
			stCapSorterWrite.bHoming 		:= NOT bCapSorterDisable; //TRUE;		
			VIS.bCapPuttedCheckHoming		:= NOT P09_CapPuttedCheck.fbCapPuttedCheck.bHomingDone AND bCapPuttedCheckEnable;
			
			//Bazowanie zakręcarki
            VIS.bGripperScrewerHoming        :=( NOT P10_GripperScrewer.fbGripperScrewer1CatchStation.bHomingDone OR
												NOT P10_GripperScrewer.fbGripperScrewer2CatchStation.bHomingDone OR
												NOT P10_GripperScrewer.fb2GripperScrewer1.bHomingDone OR
                                                NOT P10_GripperScrewer.fb2GripperScrewer2.bHomingDone) AND 
												(bGripperScrewer1Enable OR bGripperScrewer2Enable);
												
			// Bazowanie chwytaków ode zakręcarki						
			GVL.bGripperScrewerCatch1Homing := (NOT P10_GripperScrewer.fbGripperScrewer1CatchStation.bHomingDone OR
												NOT P10_GripperScrewer.fbGripperScrewer2CatchStation.bHomingDone) AND
												(bGripperScrewer1Enable OR bGripperScrewer2Enable);
			
			VIS.bBottleDragingStationHoming:= NOT P10_GripperScrewer.fbGripperScrewersDragStation.bHomingDone AND bBottleDragingStationEnable;

			// Bazowanie stacji sprawdzania nakrętek
			VIS.bCapCorrectCheckHoming 		:=	NOT P11_CapCorrectCheck.fbCapCorrectCheck.bHomingDone AND bCapCorrectCheckEnable;
			
			//Bazowanie robota
			VIS.bBottleTransferHoming		:= NOT P13_BottleTransfer.fbBottleTransfer.bHomingDone AND bBottleTransferEnable;
	
		iHomingCase										:= 20;
		
	20:
		ACT_PositioningLogic();
		
		IF NOT bAtLeastOneOfTheStationsNeedHoming AND NOT bHomingIsOnAtLeastOneStation  AND toniHomingCase20.Q THEN
			bHomingCanceled						:= FALSE;
			bRecipeChangePositioning 			:= FALSE;
			bFirstPositioningDone    			:= TRUE;
			bHoming                  			:= FALSE;
			VIS.bChooseRecipe					:= FALSE;


			ACT_ResetCommandsHoming();
			iTestiHomingCase	:=	iTestiHomingCase	+	1;
			iHomingCase									:= 0;
		END_IF
	
END_CASE
END_ACTION

ACTION ACT_Mode:

CASE fbPMLModeManager.eModeStatus OF
	
	Tc3_PackML.E_PMLUnitMode.ePMLUnitMode_UNDEFINED:

		bCycleReseting 						:= TRUE; 
		bVTEMEnable 						:= TRUE; 	//Załączenie wyspy zaworowej
		bRecipeChangePositioning 			:= TRUE;
		
		fbPMLModeManager.eModeCommand		:= Tc3_PackML.E_PMLUnitMode.ePMLUnitMode_AUTOMATIC;
		fbPMLModeManager.Execute			:= TRUE;
		
	Tc3_PackML.E_PMLUnitMode.ePMLUnitMode_AUTOMATIC:
	
		bManualMode							:= FALSE;		
		ACT_ModeAutomatic();
		ACT_ModeAutomaticConfectionEnding();		
	
		
	Tc3_PackML.E_PMLUnitMode.ePMLUnitMode_MANUAL:	
		bManualMode							:= VIS.bServiceMode;
		ACT_ModeManual();
END_CASE
END_ACTION

ACTION ACT_ModeAutomatic:

CASE fbPMLAuto.ePMLState OF
	
	Tc3_PackML.E_PMLState.ePMLState_UNDEFINED:
	
		//Zachowanie po resecie gdy jest Safety
		fbPMLAuto.Abort							:= TRUE;
		fbPMLManual.Abort						:= TRUE;
	
	Tc3_PackML.E_PMLState.ePMLState_IDLE:
	
		iPhaseChangingStep						:= 0;
		bDelayAfterStart 						:= FALSE;	//Opóźnienie po rozpoczęciu konfekcji 
		bDelayAfterStartFullRegister			:= FALSE;	//Opóżnienie po starcie sprawdzaniu rejestru pod zakręcarkami
		bROPPDelayAfterStartFullRegister		:= FALSE;
		bDelayAfterStartCapSorterFullRegister 	:= FALSE;	//Opóżnienie po starcie sprawdzaniu rejestru pod sorterem nasadek
		bWickFeederDragDelayAfterStartFullRegister:= FALSE;
		bLidSealerDragDelayAfterStartFullRegister:=FALSE;
		bVTEMEnable 							:= TRUE; 	//Załączenie wyspy zaworowej	
	
		bDelayAfterStart 						:= FALSE;	//Opóźnienie po rozpoczęciu konfekcji
		bCapSorterBottleSorterAutoStart			:= FALSE;
		
		//Przejście do bazowania po wyborze receptury z wizki, czyli jeżeli się zmienił numer indeksu lub ustawiona została zmienna
		IF VIS.bChooseRecipe THEN
			iChooseRecipe := iChooseRecipe + 1;
			VIS.bChooseRecipe				:= FALSE;
			bRecipeChangePositioning 			:= TRUE;
			bHomingDialog            			:= TRUE;
			
			fbPMLAuto.Stop						:= TRUE; 
			fbPMLManual.Stop					:= TRUE;
		END_IF
		
		//Przejśćie do bazowania jeżeli wymaga tego któraś stacja
		IF (bAtLeastOneOfTheStationsNeedHoming AND NOT P00_PackML.fbbRecipeLoading.bOut) AND NOT bHomingCanceled THEN	
			bHomingDialog  						:= TRUE;
			
			fbPMLAuto.Stop						:= TRUE; 
			fbPMLManual.Stop					:= TRUE;  
		END_IF
	 
	Tc3_PackML.E_PMLState.ePMLState_STARTING:
	
	
		//Właczanie bitów przed uruchomieniem maszyny
		ACT_PhaseChanging(); //Procedura zmiany fazy (jednofazowe-dwufazowe)
		IF P00_Visualization.iCaseDialogWeighing = 0 THEN
		
			(*Usuwanie zmiennych od sprawdzania logowania*)
			VIS.bAllowStart			:= FALSE;
			VIS.bCheckStart			:= FALSE;		
			(*Wlaczanie bitów przed uruchomieniem maszyny*)
			IF bLabelMachineEnable THEN					//Wlaczanie etykieciarki jezeli jest zalaczona w recepturach
				bLabelMachineCmdStart := TRUE;
			END_IF
			IF bCapFeederEnable THEN
				VIS.bCapFeederRun := TRUE;
			END_IF	
			IF bBadBottleConveyorEnable  THEN
				bBadBottleConveyorStartTrigger:=TRUE; //Dodatkowe uruchomienie na wszelki wypadek
			END_IF	
				
			//Opoźnienie 3s, np. na miganie lampek, lub uruchamianie jakiś transporterów
			IF tonStarting.Q AND (P08_CapFeeder.eCapFeederRunningState = E_CapFeederState.eSleeveFull OR NOT bCapFeederEnable) THEN
				bDelayAfterStart					:= TRUE;		//Opóźnienie po rozpoczęciu konfekcji
				bLongDelayAfterStart				:= TRUE;		//Długie pojedyńcze opóźnienie w pierwszym ruchu po rozpoczęciu konfekcji
					
				fbPMLAuto.StateComplete				:= TRUE;
				fbPMLManual.StateComplete			:= TRUE;	
			END_IF
			
		END_IF	
		
		
	
	Tc3_PackML.E_PMLState.ePMLState_EXECUTE:
	
		ACT_CycleLogic();
		ACT_CapSorterBottleSorterAutoStart();
		bHomingCanceled				:= FALSE;
		
		//IF P16_LabelMachine.tonLabelMachineFullSensorInfo.Q THEN
		//	fbPMLAuto.Suspend			:= TRUE;	
		//	fbPMLAuto.Suspend			:= TRUE;	
		//END_IF
	
	Tc3_PackML.E_PMLState.ePMLState_SUSPENDING:
	
		ACT_CycleLogic();
		ACT_CapSorterBottleSorterAutoStart();
		fbPMLAuto.StateComplete		:= TRUE;
		fbPMLManual.StateComplete	:= TRUE;	
		
	Tc3_PackML.E_PMLState.ePMLState_SUSPENDED:
	
		ACT_CycleLogic();
		ACT_CapSorterBottleSorterAutoStart();
	
		IF NOT P16_LabelMachine.tonLabelMachineFullSensorInfo.Q THEN
			fbPMLAuto.UnSuspend		:= TRUE;	
			fbPMLAuto.UnSuspend		:= TRUE;	
		END_IF
			
	Tc3_PackML.E_PMLState.ePMLState_UNSUSPENDING:
	
		ACT_CycleLogic();
		ACT_CapSorterBottleSorterAutoStart();
		
		fbPMLAuto.StateComplete		:= TRUE;
		fbPMLManual.StateComplete	:= TRUE;	

	Tc3_PackML.E_PMLState.ePMLState_COMPLETING:
	
		ACT_CycleLogic();
		
		fbPMLAuto.StateComplete				:= TRUE;
		fbPMLManual.StateComplete			:= TRUE;	
		
	
	Tc3_PackML.E_PMLState.ePMLState_COMPLETE:
	
		;
	
	Tc3_PackML.E_PMLState.ePMLState_ABORTING:
	
		ACT_Aborting();
	
	Tc3_PackML.E_PMLState.ePMLState_ABORTED:
	
		ACT_Aborted();
	
	Tc3_PackML.E_PMLState.ePMLState_CLEARING:
	
		ACT_Clearing();
	
	Tc3_PackML.E_PMLState.ePMLState_STOPPING:
	
		VIS.bConfectionEnding	:=	FALSE;
		ACT_Stopping();
	
	Tc3_PackML.E_PMLState.ePMLState_STOPPED:
	
		ACT_Stopped();
	
	Tc3_PackML.E_PMLState.ePMLState_RESETTING:
	
		ACT_Resetting();
END_CASE
END_ACTION

ACTION ACT_ModeAutomaticConfectionEnding:
tonFormPresent(IN:=P00_ReadRFIDCard.IbDispencerReaderTagPresent AND (NOT MAIN.IbBottleInFormCheckBottleSensor), pt:=T#210MS);

IF vis.bConfectionEnding THEN
	IF tonFormPresent.q AND(NOT MAIN.IbBottleInFormCheckBottleSensor) AND diRFIDNumberFormatDispencerConfectionEnd =0 AND diPreviouslyReaded<>P00_ReadRFIDCard.fbDispencerReader.diReadedCode THEN// AND MAIN.IbFormCheckFormSensor THEN
	iEndConfectionCounter:=iEndConfectionCounter+1;
	diPreviouslyReaded:=P00_ReadRFIDCard.fbDispencerReader.diReadedCode;
		IF (iEndConfectionCounter=10) THEN
		diRFIDNumberFormatDispencerConfectionEnd:=P00_ReadRFIDCard.fbDispencerReader.diReadedCode;
		END_IF
	END_IF		
END_IF

IF P00_ReadRFIDCard.fbBottleTransferReader.diReadedCode=diRFIDNumberFormatDispencerConfectionEnd THEN
	bStartEndCofectionTimer:=TRUE;
END_IF

tonEndOfConfecion (IN:=bStartEndCofectionTimer, PT:=T#5S);

IF NOT vis.bConfectionEnding THEN
	bStartEndCofectionTimer:=FALSE;
	diRFIDNumberFormatDispencerConfectionEnd:=0;
	iEndConfectionCounter:=0;
	diPreviouslyReaded:=0;
END_IF
END_ACTION

ACTION ACT_ModeManual:

CASE fbPMLManual.ePMLState OF
	
	 Tc3_PackML.E_PMLState.ePMLState_IDLE:
	 
	 	//Na conajmniej jednej ze stacji włączono bazowanie
		IF (bHomingIsOnAtLeastOneStation AND NOT bHomingCanceled) OR rtHomingIsOnAtLeastOneStation.Q THEN
			bHomingDialog  							:= TRUE;
			fbPMLAuto.Stop							:= TRUE; 
			fbPMLManual.Stop						:= TRUE;
		END_IF

	 
	Tc3_PackML.E_PMLState.ePMLState_ABORTING:

		ACT_Aborting();

	Tc3_PackML.E_PMLState.ePMLState_ABORTED: 
	
		ACT_Aborted();
		
	Tc3_PackML.E_PMLState.ePMLState_CLEARING:
	
		ACT_Clearing();
		
	Tc3_PackML.E_PMLState.ePMLState_STOPPING:
	
		ACT_Stopping(); {warning 'USUNĄĆ STOPPING W MANUALU ŻEBY NIE WYCHODZIŁO Z MANUALA?"}
		
	Tc3_PackML.E_PMLState.ePMLState_STOPPED:
	
		ACT_Stopped(); {warning 'USUNĄĆ STOPPING W MANUALU ŻEBY NIE WYCHODZIŁO Z MANUALA?"}
		
	Tc3_PackML.E_PMLState.ePMLState_RESETTING:
	
		ACT_Resetting();
END_CASE
END_ACTION

ACTION ACT_PhaseChanging:
(*
Nazwa:			ACT_PhaseChanging
Opis:			
Wersja:			v0.1
Data:			2022-05-26
Autor:			DP
Urzadzenia:		
Konfiguracja:	
Info: 
- Wywoływanie w Starting, Execute, Stopping
- Wykrywanie przełączenia dwufazy
- Blokowanie szlabanu przed dozownikami
*)

bPhaseChanging;	
tonLongDelayFirstDraging;




(********Wykrywanie przełączenia*********)
IF P00_PackML.fbPMLAuto.ePMLState = E_PMLState.ePMLState_STARTING THEN
	IF NOT bDosingTwoPhases AND VIS.bDosingTwoPhasesShow AND NOT bPhaseChanging THEN
		bCycleReseting			:=	TRUE;
		bPhaseChanging			:=	TRUE;
	END_IF
	IF bDosingTwoPhases AND NOT VIS.bDosingTwoPhasesShow AND NOT bPhaseChanging THEN
		bCycleReseting			:=	TRUE;
		bPhaseChanging			:=	TRUE;
	END_IF
END_IF
(****************************************)


tonNotLongDelayAfterStart(IN:= bPhaseChanging AND iPhaseChangingStep=30 AND NOT bLongDelayAfterStart, PT:=T#5S);

IF tonNotLongDelayAfterStart.Q THEN
	bLongDelayAfterStart:=TRUE;
END_IF


(****Procedura przełączania fazy*********)
tonPhaseChangingCase110Delay	(IN:=iPhaseChangingStep=110	OR iPhaseChangingStep=130 ,PT:=T#3S);
tonPhaseChangingCase200Delay	(IN:=iPhaseChangingStep=200,PT:=T#3S);
tonPhaseChangingCase210Delay	(IN:=iPhaseChangingStep=210	OR iPhaseChangingStep=240  OR iPhaseChangingStep=260 OR iPhaseChangingStep=280	OR iPhaseChangingStep=300,PT:=T#3S);

CASE iPhaseChangingStep OF
	
	0:
		IF bPhaseChanging AND NOT (P00_PackML.fbPMLAuto.ePMLState = E_PMLState.ePMLState_STOPPING) AND (P00_PackML.fbPMLAuto.ePMLState = Tc3_PackML.E_PMLState.ePMLState_EXECUTE) THEN
			iPhaseChangingStep						:=	iPhaseChangingStep	+	10;	
		END_IF
			
	10:
		eBeforeDispencersPackageState[1]			:=	eClearPackageState;
		eBeforeDispencersPackageState[2]			:=	eClearPackageState;		
		eBeforeDispencersPackageState[3]			:=	eClearPackageState;			
		eBeforeDispencersPackageState[4]			:=	eClearPackageState;	
                                                    
		eDispencersPackageState[1]					:=	eClearPackageState;
		eDispencersPackageState[2]					:=	eClearPackageState;		
		eDispencersPackageState[3]					:=	eClearPackageState;			
		eDispencersPackageState[4]					:=	eClearPackageState;
                                                    
		eAfterDispencersPackageState[1]				:=	eClearPackageState;
		eAfterDispencersPackageState[2]				:=	eClearPackageState;		
		eAfterDispencersPackageState[3]				:=	eClearPackageState;			
		eAfterDispencersPackageState[4]				:=	eClearPackageState;	
	
		eWeightPackageState[4]						:=	eClearPackageState;	
		eWeightPackageState[3]						:=	eClearPackageState;	
		eWeightPackageState[2]						:=	eClearPackageState;	
		eWeightPackageState[1]						:=	eClearPackageState;	
                                           
		eBeforeDispencer12PackageState2Phase[1]		:=	eClearPackageState;
		eBeforeDispencer12PackageState2Phase[2]		:=	eClearPackageState;	                           				
		eDispencer12PackageState2Phase[1]			:=	eClearPackageState;	
		eDispencer12PackageState2Phase[2]			:=	eClearPackageState;
		eAfterDispencer12PackageState2Phase[1]		:=	eClearPackageState;
		eAfterDispencer12PackageState2Phase[2]		:=	eClearPackageState;			
		                                            
		eBeforeDispencer34PackageState2Phase[1]		:=  eClearPackageState;
		eBeforeDispencer34PackageState2Phase[2]		:=	eClearPackageState;
		eDispencer34PackageState2Phase[1]			:=	eClearPackageState;
		eDispencer34PackageState2Phase[2]			:=	eClearPackageState;		
		eAfterDispencer34PackageState2Phase[1]		:=	eClearPackageState;	
		eAfterDispencer34PackageState2Phase[2]		:=	eClearPackageState;

		eWeightPackage2PhasePackageState[2]			:=	eClearPackageState;
		eWeightPackage2PhasePackageState[1]			:=	eClearPackageState;
	
		
		iPhaseChangingStep							:=	iPhaseChangingStep	+	10;	
		
	20: 
		IF tonDelayAfterStart.Q THEN //3s po starcie
			iPhaseChangingStep						:=	iPhaseChangingStep	+	10;	
		END_IF
		
	30:
		fbIbFourthFormCheckFormSensor.bOut;			
		fbIbTwoPhasesFormSensorBetweenDispencers.bOut;	
		fbIbSecondFormCheckFormSensor.bOut;
		P05_Weight.IbWeight6FormSensor;			
		P02_Dispencers.fbDispencersDragLeftStation.bCycleDone;
		P02_Dispencers.fbDispencersDragRightStation.bCycleDone;		
		VIS.bFormsDragingLeftRun;	
		VIS.bFormsDragingRightRun;		
		
		IF NOT bDosingTwoPhases THEN
			iPhaseChangingStep						:=	100;
		ELSE
			iPhaseChangingStep						:=	200;
		END_IF
		
	100: //Przełączenie na jednofaza -> dwufaze
		IF	NOT fbIbTwoPhasesFormSensorBetweenDispencers.bOut AND
			NOT P05_Weight.IbWeight4FormSensor AND 
			NOT P00_ReadRFIDCard.bReadedCardAfterDispencers
		 THEN
			VIS.bFormsDragingLeftRun 				:=	TRUE;
			VIS.bFormsDragingRightRun				:=	TRUE;
		END_IF
		
		IF 	P02_Dispencers.fbDispencersDragLeftStation.bCycleDone AND P02_Dispencers.fbDispencersDragRightStation.bCycleDone THEN
			VIS.bFormsDragingLeftRun 				:=	FALSE;
			VIS.bFormsDragingRightRun				:=	FALSE;				
			iPhaseChangingStep						:=	iPhaseChangingStep	+	10;	
		END_IF	
		
	110:
		IF tonPhaseChangingCase110Delay.Q THEN
			//P06_LidFeeder.QbLidFeederDragActuator	:=FALSE;
			iPhaseChangingStep						:=	iPhaseChangingStep	+	10;	
		END_IF	
		
	120:
		IF	NOT fbIbTwoPhasesFormSensorBetweenDispencers.bOut AND
			NOT P05_Weight.IbWeight4FormSensor AND 
			NOT P00_ReadRFIDCard.bReadedCardAfterDispencers
		 THEN
		 	//P06_LidFeeder.bMovetoEndPositionLidFeeder				:=	TRUE;
			VIS.bFormsDragingLeftRun 				:=	TRUE;
			VIS.bFormsDragingRightRun				:=	TRUE;
		END_IF
		
		IF 	P02_Dispencers.fbDispencersDragLeftStation.bCycleDone AND P02_Dispencers.fbDispencersDragRightStation.bCycleDone THEN
			VIS.bFormsDragingLeftRun 				:=	FALSE;
			VIS.bFormsDragingRightRun				:=	FALSE;				
			iPhaseChangingStep						:=	iPhaseChangingStep	+	10;	
		END_IF	
		
	130:
		IF tonPhaseChangingCase110Delay.Q THEN
			//VIS.bLidFeederDragingStationRun	:=TRUE;
			iPhaseChangingStep						:=	iPhaseChangingStep	+	10;	
		END_IF	

	140:
		iPhaseChangingStep							:=	iPhaseChangingStep	+	10;
	150:
		
		bDosingTwoPhases							:= 	TRUE;
		iPhaseChangingStep							:=	500	;
		
		
	200: //Przełączenie na dwufaza -> jednofaza	
		//P06_LidFeeder.QbLidFeederDragActuator	:=TRUE;		
		IF	tonPhaseChangingCase200Delay.Q AND
			NOT fbIbSecondFormCheckFormSensor.bOut AND
			NOT	P05_Weight.IbWeight6FormSensor AND
			NOT P00_ReadRFIDCard.bReadedCardAfterDispencers2Phase 
		 THEN
			VIS.bFormsDragingLeftRun 				:=	TRUE;
		END_IF
		
		IF 	P02_Dispencers.fbDispencersDragLeftStation.bCycleDone THEN
			VIS.bFormsDragingLeftRun 				:=	FALSE;		
			iPhaseChangingStep						:=	iPhaseChangingStep	+	10;	
		END_IF	
	210:
	
		IF tonPhaseChangingCase210Delay.Q THEN
			iPhaseChangingStep						:=	iPhaseChangingStep	+	10;	
		END_IF
		
	220:
		IF fbIbTwoPhasesFormSensorBetweenDispencers.bOut THEN //Jeżeli są jeszcze jakies formatki
			iPhaseChangingStep						:=	200;
		ELSE
			iPhaseChangingStep						:=	iPhaseChangingStep	+	10;	
		END_IF
		
	230:
	
		VIS.bFormsDragingRightRun 					:=	TRUE;	
		IF 	P02_Dispencers.fbDispencersDragRightStation.bCycleDone THEN
			VIS.bFormsDragingRightRun 				:=	FALSE;		
			iPhaseChangingStep						:=	iPhaseChangingStep	+	10;	
		END_IF	
		
	240:
		IF tonPhaseChangingCase210Delay.Q THEN
			iPhaseChangingStep						:=	iPhaseChangingStep	+	10;	
		END_IF
		
	250:
		VIS.bFormsDragingRightRun 					:=	TRUE;	
		IF 	P02_Dispencers.fbDispencersDragRightStation.bCycleDone THEN
			VIS.bFormsDragingRightRun 				:=	FALSE;		
			iPhaseChangingStep						:=	iPhaseChangingStep	+	10;	
		END_IF	
		
	260:	
		IF tonPhaseChangingCase210Delay.Q THEN
			iPhaseChangingStep						:=	iPhaseChangingStep	+	10;	
		END_IF
		
	270:	
		IF	NOT fbIbSecondFormCheckFormSensor.bOut AND
			NOT	P05_Weight.IbWeight6FormSensor AND
			NOT P00_ReadRFIDCard.bReadedCardAfterDispencers2Phase 
		 THEN
			VIS.bFormsDragingLeftRun 				:=	TRUE;
		END_IF
		
		IF 	P02_Dispencers.fbDispencersDragLeftStation.bCycleDone THEN
			VIS.bFormsDragingLeftRun 				:=	FALSE;		
			iPhaseChangingStep						:=	iPhaseChangingStep	+	10;	
		END_IF	
		
	280:	
		IF tonPhaseChangingCase210Delay.Q THEN
			iPhaseChangingStep						:=	iPhaseChangingStep	+	10;	
		END_IF
		
	290:
		IF	NOT fbIbSecondFormCheckFormSensor.bOut AND
			NOT	P05_Weight.IbWeight6FormSensor AND
			NOT P00_ReadRFIDCard.bReadedCardAfterDispencers2Phase 
		 THEN
			VIS.bFormsDragingLeftRun 				:=	TRUE;
		END_IF
		
		IF 	P02_Dispencers.fbDispencersDragLeftStation.bCycleDone THEN
			VIS.bFormsDragingLeftRun 				:=	FALSE;		
			iPhaseChangingStep						:=	iPhaseChangingStep	+	10;	
		END_IF	
		
	300:	
		IF tonPhaseChangingCase210Delay.Q THEN
			iPhaseChangingStep						:=	iPhaseChangingStep	+	10;	
		END_IF
		
	310:
		IF	NOT fbIbSecondFormCheckFormSensor.bOut AND
			NOT	P05_Weight.IbWeight6FormSensor AND
			NOT P00_ReadRFIDCard.bReadedCardAfterDispencers2Phase 
		 THEN
			VIS.bFormsDragingLeftRun 				:=	TRUE;
		END_IF
		
		IF 	P02_Dispencers.fbDispencersDragLeftStation.bCycleDone THEN
			VIS.bFormsDragingLeftRun 				:=	FALSE;		
			iPhaseChangingStep						:=	iPhaseChangingStep	+	10;	
			//iPhaseChangingStep						:=	iPhaseChangingStep	+	5;	
		END_IF		
	//vasyl
	315:
		IF NOT MAIN.IbLidSealerAfterSensor	THEN
			VIS.bLidSealerDragingStationRun:=TRUE;
		END_IF
		IF 	P06_LidSealer.fbLidSealerDragStation.bCycleDone THEN
			VIS.bLidSealerDragingStationRun:=FALSE;
			iPhaseChangingStep						:=	iPhaseChangingStep	+	5;
		END_IF
		
	320:
		bDosingTwoPhases							:= 	FALSE;
		iPhaseChangingStep							:=	500;
		
	500: //Koniec
		IF	NOT fbIbTwoPhasesFormSensorBetweenDispencers.bOut AND
			NOT P05_Weight.IbWeight4FormSensor AND 
			NOT P00_ReadRFIDCard.bReadedCardAfterDispencers AND
			
			NOT	fbIbTwoPhasesFormSensorBetweenDispencers.bOut AND 	
			NOT fbIbSecondFormCheckFormSensor.bOut AND
			NOT	P05_Weight.IbWeight6FormSensor AND
			NOT P00_ReadRFIDCard.bReadedCardAfterDispencers2Phase 
		 THEN			
			iPhaseChangingStep						:=	iPhaseChangingStep	+	10;	
		END_IF

	510:

		eBeforeDispencersPackageState[1]			:=	eClearPackageState;
		eBeforeDispencersPackageState[2]			:=	eClearPackageState;		
		eBeforeDispencersPackageState[3]			:=	eClearPackageState;			
		eBeforeDispencersPackageState[4]			:=	eClearPackageState;	
                                                    
		eDispencersPackageState[1]					:=	eClearPackageState;
		eDispencersPackageState[2]					:=	eClearPackageState;		
		eDispencersPackageState[3]					:=	eClearPackageState;			
		eDispencersPackageState[4]					:=	eClearPackageState;
                                                    
		eAfterDispencersPackageState[1]				:=	eClearPackageState;
		eAfterDispencersPackageState[2]				:=	eClearPackageState;		
		eAfterDispencersPackageState[3]				:=	eClearPackageState;			
		eAfterDispencersPackageState[4]				:=	eClearPackageState;
	
		eWeightPackageState[4]						:=	eClearPackageState;	
		eWeightPackageState[3]						:=	eClearPackageState;	
		eWeightPackageState[2]						:=	eClearPackageState;	
		eWeightPackageState[1]						:=	eClearPackageState;	
		                                            
		eBeforeDispencer12PackageState2Phase[1]		:=	eClearPackageState;
		eBeforeDispencer12PackageState2Phase[2]		:=	eClearPackageState;	                           				
		eDispencer12PackageState2Phase[1]			:=	eClearPackageState;	
		eDispencer12PackageState2Phase[2]			:=	eClearPackageState;
		eAfterDispencer12PackageState2Phase[1]		:=	eClearPackageState;
		eAfterDispencer12PackageState2Phase[2]		:=	eClearPackageState;			
		                                            
		eBeforeDispencer34PackageState2Phase[1]		:=  eClearPackageState;
		eBeforeDispencer34PackageState2Phase[2]		:=	eClearPackageState;
		eDispencer34PackageState2Phase[1]			:=	eClearPackageState;
		eDispencer34PackageState2Phase[2]			:=	eClearPackageState;		
		eAfterDispencer34PackageState2Phase[1]		:=	eClearPackageState;	
		eAfterDispencer34PackageState2Phase[2]		:=	eClearPackageState;

		eWeightPackage2PhasePackageState[2]			:=	eClearPackageState;
		eWeightPackage2PhasePackageState[1]			:=	eClearPackageState;
		
		iPhaseChangingStep							:=	600;
		
	600:
		bPhaseChanging								:=	FALSE;		
		
END_CASE
(****************************************)
END_ACTION

ACTION ACT_PmlChangeMode:

CASE iChangeModeStep OF
	
	0:
		//Sprawdzam czy mam Manual
		IF VIS.bServiceMode THEN
			
			IF fbPMLModeManager.eModeStatus <> Tc3_PackML.E_PMLUnitMode.ePMLUnitMode_MANUAL THEN
				iChangeModeStep				:= 200;
			END_IF
		
		ELSE
			
			IF fbPMLModeManager.eModeStatus <> Tc3_PackML.E_PMLUnitMode.ePMLUnitMode_AUTOMATIC THEN
				iChangeModeStep				:= 100;
			END_IF
		
		END_IF
	
	100: //Auto
	
		IF NOT bHomingDialog AND bHoming THEN
			bHoming	:= FALSE;
		END_IF
	
		IF fbPMLAuto.ePMLState = Tc3_PackML.E_PMLState.ePMLState_IDLE OR fbPMLAuto.ePMLState = Tc3_PackML.E_PMLState.ePMLState_STOPPED OR fbPMLAuto.ePMLState = Tc3_PackML.E_PMLState.ePMLState_ABORTED OR
			fbPMLAuto.ePMLState = Tc3_PackML.E_PMLState.ePMLState_HELD OR fbPMLAuto.ePMLState = Tc3_PackML.E_PMLState.ePMLState_SUSPENDED OR fbPMLAuto.ePMLState = Tc3_PackML.E_PMLState.ePMLState_COMPLETE THEN
			
			fbPMLModeManager.eModeCommand					:= Tc3_PackML.E_PMLUnitMode.ePMLUnitMode_AUTOMATIC;
			fbPMLModeManager.Execute						:= TRUE;
			iChangeModeStep									:= 300;
		ELSE	
			fbPMLModeManager.Execute						:= FALSE;
		END_IF
		
		IF fbPMLModeManager.Error THEN
			iChangeModeStep									:= 300;
		END_IF
	
	200: //Manual
	
		IF fbPMLAuto.ePMLState = Tc3_PackML.E_PMLState.ePMLState_IDLE OR fbPMLAuto.ePMLState = Tc3_PackML.E_PMLState.ePMLState_STOPPED OR fbPMLAuto.ePMLState = Tc3_PackML.E_PMLState.ePMLState_ABORTED OR
			fbPMLAuto.ePMLState = Tc3_PackML.E_PMLState.ePMLState_HELD OR fbPMLAuto.ePMLState = Tc3_PackML.E_PMLState.ePMLState_SUSPENDED OR fbPMLAuto.ePMLState = Tc3_PackML.E_PMLState.ePMLState_COMPLETE THEN
			
			fbPMLModeManager.eModeCommand					:= Tc3_PackML.E_PMLUnitMode.ePMLUnitMode_MANUAL;
			fbPMLModeManager.Execute						:= TRUE;
			iChangeModeStep									:= 300;
		ELSE	
			fbPMLModeManager.Execute						:= FALSE;
		END_IF
		
		IF fbPMLModeManager.Error THEN
			iChangeModeStep									:= 300;
		END_IF
	
	300:
		IF fbPMLModeManager.Done OR fbPMLModeManager.Error THEN
			ACT_ResetCommands();
			iChangeModeStep									:= 0;
			fbPMLModeManager.Execute						:= FALSE;
		END_IF
		
END_CASE
END_ACTION

ACTION ACT_PmlModeManager:


IF fbPMLModeManager.eModeStatus = Tc3_PackML.E_PMLUnitMode.ePMLUnitMode_AUTOMATIC THEN
	fbPMLModeManager.ePMLState		:= fbPMLAuto.ePMLState;
END_IF

IF fbPMLModeManager.eModeStatus = Tc3_PackML.E_PMLUnitMode.ePMLUnitMode_MANUAL THEN
	fbPMLModeManager.ePMLState		:= fbPMLManual.ePMLState;
END_IF

// Zarządzanie trybami - PackML ModeManager

fbPMLModeManager(
	Execute:= , 
	eModeCommand:= , 
	ePMLState:= , 
	eModeStatus=> , 
	Done=> , 
	Error=> , 
	ErrorID=> );
END_ACTION

ACTION ACT_PmlResetCommands:


// Auto
fbPMLAuto.Start				:= FALSE;
fbPMLAuto.Hold				:= FALSE;
fbPMLAuto.UnHold			:= FALSE;
fbPMLAuto.Suspend			:= FALSE;
fbPMLAuto.UnSuspend			:= FALSE;
fbPMLAuto.Abort				:= FALSE;
fbPMLAuto.Stop				:= FALSE;
fbPMLAuto.Complete			:= FALSE;
fbPMLAuto.Clear				:= FALSE;
fbPMLAuto.Reset				:= FALSE;
fbPMLAuto.StateComplete		:= FALSE;


// Manual
fbPMLManual.Start			:= FALSE;
fbPMLManual.Hold			:= FALSE;
fbPMLManual.UnHold			:= FALSE;
fbPMLManual.Suspend			:= FALSE;
fbPMLManual.UnSuspend		:= FALSE;
fbPMLManual.Abort			:= FALSE;
fbPMLManual.Stop			:= FALSE;
fbPMLManual.Complete		:= FALSE;
fbPMLManual.Clear			:= FALSE;
fbPMLManual.Reset			:= FALSE;
fbPMLManual.StateComplete	:= FALSE;


// Mode Manager				
fbPMLModeManager.Execute	:= FALSE;
END_ACTION

ACTION ACT_PmlStates:
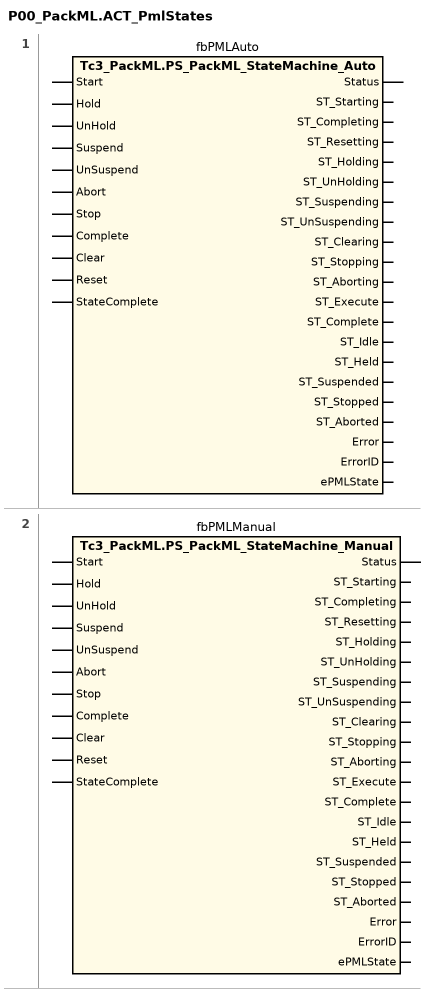
// NETWORK 1
fbPMLAuto(); // Tc3_PackML.PS_PackML_StateMachine_Auto

// NETWORK 2
fbPMLManual(); // Tc3_PackML.PS_PackML_StateMachine_Manual
END_ACTION

ACTION ACT_PositioningLogic:
(****************************************)
(** Procedura bazowania podajnika butelek**)
(****P01_BottleFeeder*******)
IF VIS.bBottleFeederHoming THEN
	GVL.bBottleFeederEnable				:=TRUE; //Włączenie stacji i kasowanie istniejacych rozkazów
	VIS.bBottleFeederRun				:=FALSE;
	bBottleFeederDoHoming :=NOT bBottleFeederHommed;
	IF bBottleFeederHommed THEN
		IF P01_BottleFeeder.fbBottleFeeder.eState=E_Station.eHomingDone THEN
			VIS.bBottleFeederHoming		:=FALSE;
			bBottleFeederHommed			:=FALSE;
		END_IF
	ELSIF 
		P01_BottleFeeder.fbBottleFeeder.eState=E_Station.eHomingDone THEN
		bBottleFeederHommed			:=TRUE;
	END_IF;
END_IF

(** Procedura bazowania podajnika opakowań**)
(****P01_PucksInserter*******)
IF VIS.bPucksInserterHoming THEN
	GVL.bPucksInserterEnable			:=TRUE; //Włączenie stacji i kasowanie istniejacych rozkazów
	VIS.bPucksInserterRun				:=FALSE;
	bPucksInserterDoHoming :=NOT bPucksInserterHommed;
	IF bPucksInserterHommed THEN
		VIS.bPucksInserterHeightSet	:=	TRUE;
		IF P01_PucksInserter.fbPucksInserter.eState=E_Station.eHomingDone THEN
			VIS.bPucksInserterHeightSet		:=FALSE;
			bPucksInserterHommed			:=FALSE;	
			bPucksInserterDoHoming 			:=FALSE;	
			VIS.bPucksInserterHoming		:=FALSE;
		END_IF
	ELSIF 	P01_PucksInserter.fbPucksInserter.eState=E_Station.eHomingDone THEN
		bPucksInserterDoHoming 				:=FALSE;
		bPucksInserterHommed				:=TRUE;
	END_IF;
END_IF


(** Procedura bazowania sortera butelek*)
tonBottleSorterHomingAndDone (IN:= stBottleSorterWrite.bHoming, PT:=T#5S);
IF tonBottleSorterHomingAndDone.Q THEN
	IF stBottleSorterRead.bHomingDone THEN
		stBottleSorterWrite.bHoming 		:= FALSE;
	END_IF	
END_IF

(******	Procedura bazowania stacji przeciągania	******)
(******	P02_Dispencers	******)
IF VIS.bFormsDragingRightHoming THEN
	GVL.bFormsDragingRightEnable:=TRUE; (*Włączenie enabla i kasowanie rozkazów*)
	VIS.bFormsDragingRightRun:=FALSE;
	GVL.bFormsDragingRightPrepareRun:=FALSE;
	bFormsDragingRightDoHoming:=NOT bFormsDragRightStationHommed;
	IF bFormsDragRightStationHommed THEN
		IF P02_Dispencers.fbDispencersDragRightStation.eState=E_Station.eHomingDone THEN
			VIS.bFormsDragingRightHoming:=FALSE;
			bFormsDragRightStationHommed:=FALSE;
		END_IF
	ELSIF P02_Dispencers.fbDispencersDragRightStation.eState=E_Station.eHomingDone THEN
			bFormsDragRightStationHommed:=TRUE;
	END_IF
END_IF


IF VIS.bFormsDragingLeftHoming THEN
	GVL.bFormsDragingLeftEnable:=TRUE; (*Włączenie enabla i kasowanie rozkazów*)
	VIS.bFormsDragingLeftRun:=FALSE;
	GVL.bFormsDragingLeftPrepareRun:=FALSE;
	bFormsDragingLeftDoHoming:=NOT bFormsDragLeftStationHommed;
	IF bFormsDragLeftStationHommed THEN
		IF P02_Dispencers.fbDispencersDragLeftStation.eState=E_Station.eHomingDone THEN
			VIS.bFormsDragingLeftHoming:=FALSE;
			bFormsDragLeftStationHommed:=FALSE;
		END_IF
	ELSIF P02_Dispencers.fbDispencersDragLeftStation.eState=E_Station.eHomingDone THEN
			bFormsDragLeftStationHommed:=TRUE;
	END_IF
END_IF


(****************************************)

(*******P02_Dispencers******)
(****** Procedura bazowania dozowników,podnosnika chwytaka i tacki dozownika******)

IF VIS.bDispencersHoming THEN
	VIS.bDispencer1Dose:=VIS.bDispencer2Dose:=VIS.bDispencer3Dose:=VIS.bDispencer3Dose:=VIS.bDispencer4Dose:=FALSE;
	bDispencer1Enable:=bDispencer2Enable:=bDispencer3Enable:=bDispencer4Enable:=TRUE;
	bDispencersDoHoming:=NOT bDispencersHommed;
	IF bDispencersHommed THEN	
		VIS.bDispencersCatchHeightSet:=TRUE;
		IF P02_Dispencers.fbDispencersCatch1Station.eState=E_Station.eHomingDone AND P02_Dispencers.fbDispencersCatch2Station.eState=E_Station.eHomingDone 
		AND P02_Dispencers.fbDispencersCatch3Station.eState=E_Station.eHomingDone AND P02_Dispencers.fbDispencersCatch4Station.eState=E_Station.eHomingDone THEN
		
			VIS.bDispencer12LifterHeightSet:=VIS.bDispencer34LifterHeightSet:=TRUE;
			
			IF	P02_Dispencers.fbDispencer1.eState=E_Station.eHomingDone AND P02_Dispencers.fbDispencer2.eState=E_Station.eHomingDone AND 
				P02_Dispencers.fbDispencer3.eState=E_Station.eHomingDone AND P02_Dispencers.fbDispencer4.eState=E_Station.eHomingDone THEN
				VIS.bDispencer12LifterHeightSet:=VIS.bDispencer34LifterHeightSet:=FALSE;
				VIS.bDispencersCatchHeightSet:=FALSE;
				bDispencersHommed:=FALSE;
				VIS.bDispencersHoming:=FALSE;
			END_IF
		END_IF
	ELSIF NOT bDispencersHommed AND P02_Dispencers.fbDispencer1.eState=E_Station.eHomingDone AND P02_Dispencers.fbDispencer2.eState=E_Station.eHomingDone AND
									P02_Dispencers.fbDispencer3.eState=E_Station.eHomingDone AND P02_Dispencers.fbDispencer4.eState=E_Station.eHomingDone THEN
		bDispencersCatch1DoHoming:=bDispencersCatch2DoHoming:=bDispencersCatch3DoHoming:=bDispencersCatch4DoHoming:=TRUE;
		IF P02_Dispencers.fbDispencersCatch1Station.eState=E_Station.eHomingDone AND P02_Dispencers.fbDispencersCatch2Station.eState=E_Station.eHomingDone 
		AND P02_Dispencers.fbDispencersCatch3Station.eState=E_Station.eHomingDone AND P02_Dispencers.fbDispencersCatch4Station.eState=E_Station.eHomingDone THEN
			bDispencersDoHoming:=FALSE;
			bDispencersCatch1DoHoming:=bDispencersCatch2DoHoming:=bDispencersCatch3DoHoming:=bDispencersCatch4DoHoming:=FALSE;
			bDispencersHommed:=TRUE;
		END_IF
	END_IF
END_IF
(****************************************)

(****************************************)

(******	Procedura bazowania stacji podnoszenia formatek	******)
(****** 	P05_Weight	  *****)

IF VIS.bWeightLiftHoming THEN

	IF (NOT bDosingTwoPhases AND P05_Weight.fbWeightStation.bHomingDone) OR  (bDosingTwoPhases AND P05_Weight.fbWeightStation2Phase.bHomingDone) THEN
		bWeightLiftHommed					:= FALSE;
		GVL.bWeightLiftDoHoming				:= FALSE;
		VIS.bWeightLiftHoming				:= FALSE;
		GVL.bWeightLiftEnable				:= TRUE;
		iii									:= iii+1;
	END_IF
	IF NOT P05_Weight.fbWeightStation.bHomingDone OR (NOT P05_Weight.fbWeightStation2Phase.bHomingDone AND bDosingTwoPhases) THEN
		GVL.bWeightLiftEnable					:= TRUE; 
		GVL.bWeightLiftDoHoming					:= TRUE;
	END_IF
	
ELSE
	IF P05_Weight.fbWeightStation.bHomingDone AND (P05_Weight.fbWeightStation2Phase.bHomingDone OR NOT bDosingTwoPhases) THEN
		bWeightLiftHommed					:= FALSE;
		VIS.bWeightLiftRun					:= FALSE;
		bWeightLift2PhaseRun				:= FALSE;
		GVL.bWeightLiftEnable				:= TRUE;
		GVL.bWeightLiftDoHoming				:= FALSE;
	END_IF
	//VIS.bWeightLiftRun						:= FALSE;
	//GVL.bWeightLiftEnable					:= TRUE; (*Włączenie enabla i kasowanie rozkazów*)
	//GVL.bWeightLiftDoHoming					:= TRUE;
		
END_IF
(*****P06_WickFeeder********)
(******* Procedura bazowania stacji********)
IF VIS.bWickFeederHoming THEN
	bWickFeederEnable:=TRUE;
	bWickFeederDoHoming:=NOT bWickFeederHommed;
	IF bWickFeederHommed THEN
		VIS.bWickFeederHeightSet:=TRUE;
		IF P06_WickFeeder.fbWickFeederSt.eState=E_Station.eHomingDone   THEN
			VIS.bWickFeederHeightSet:=FALSE;
			bWickFeederHommed:=FALSE;
			bWickFeederDoHoming:=FALSE;
			VIS.bWickFeederHoming:=FALSE;
		END_IF
	ELSIF P06_WickFeeder.fbWickFeederSt.eState=E_Station.eHomingDone  THEN
			bWickFeederDoHoming:=FALSE;
			bWickFeederHommed:=TRUE;
	END_IF
END_IF

IF VIS.bWickFeederDragingHoming THEN
	bWickFeederDragingStationEnable:=TRUE;
	bWickFeederDragingStationDoHoming:=NOT bWickFeederDragingHommed;
	IF bWickFeederDragingHommed THEN
		IF P06_WickFeeder.fbWickFeederDragStation.eState=E_Station.eHomingDone THEN
			bWickFeederDragingHommed:=FALSE;
			bWickFeederDragingStationDoHoming:=FALSE;
			VIS.bWickFeederDragingHoming:=FALSE;
		END_IF
	ELSIF P06_WickFeeder.fbWickFeederDragStation.eState=E_Station.eHomingDone THEN
			bWickFeederDragingHommed:=TRUE;
	END_IF
END_IF

(*****P06_LidFeeder********)
(******* Procedura bazowania stacji********)
IF VIS.bLidFeederHoming THEN
	bLidFeederEnable:=TRUE;
	bLidFeederDoHoming:=NOT bLidFeederHommed;
	IF bLidFeederHommed THEN
		VIS.bLidFeederHeightSet:=TRUE;
		IF P06_LidFeeder.fbLidFeeder.eState=E_Station.eHomingDone AND P06_LidFeeder.fbLidFeeder2.eState=E_Station.eHomingDone  THEN
			VIS.bLidFeederHeightSet:=FALSE;
			bLidFeederHommed:=FALSE;
			bLidFeederDoHoming:=FALSE;
			VIS.bLidFeederHoming:=FALSE;
		END_IF
	ELSIF P06_LidFeeder.fbLidFeeder.eState=E_Station.eHomingDone AND P06_LidFeeder.fbLidFeeder2.eState=E_Station.eHomingDone THEN
			bLidFeederDoHoming:=FALSE;
			bLidFeederHommed:=TRUE;
	END_IF
END_IF

IF VIS.bLidFeederDragingHoming THEN
	bLidFeederDragingStationEnable:=TRUE;
	bLidFeederDragingStationDoHoming:=NOT bLidFeederDragingHommed;
	IF bLidFeederDragingHommed THEN
		IF P06_LidFeeder.fbLidFeederDragStation.eState=E_Station.eHomingDone THEN
			bLidFeederDragingHommed:=FALSE;
			bLidFeederDragingStationDoHoming:=FALSE;
			VIS.bLidFeederDragingHoming:=FALSE;
		END_IF
	ELSIF P06_LidFeeder.fbLidFeederDragStation.eState=E_Station.eHomingDone THEN
			bLidFeederDragingHommed:=TRUE;
	END_IF
END_IF

(*****P06_LidPuttedCheck********)
(******* Procedura bazowania stacji********)
(*IF VIS.bLidPuttedCheckHoming THEN
	bLidPuttedCheckEnable:=TRUE;
	bLidPuttedCheckDoHoming:=NOT bLidPuttedCheckHommed;
	IF bLidPuttedCheckHommed THEN
		VIS.bLidPuttedCheckHeightSet:=TRUE;
		IF P06_LidPuttedCheck.fbLidPuttedCheck.eState=E_Station.eHomingDone THEN
			VIS.bLidPuttedCheckHeightSet:=FALSE;
			bLidPuttedCheckHommed:=FALSE;
			bLidPuttedCheckDoHoming:=FALSE;
			VIS.bLidPuttedCheckHoming:=FALSE;
		END_IF
	ELSIF P06_LidPuttedCheck.fbLidPuttedCheck.eState=E_Station.eHomingDone THEN
			bLidPuttedCheckDoHoming:=FALSE;
			bLidPuttedCheckHommed:=TRUE;
	END_IF
END_IF*)

(*****P06_LidSealer********)
(******* Procedura bazowania stacji********)
IF VIS.bLidSealerHoming THEN
	bLidSealerEnable:=TRUE;
	bLidSealerDoHoming:=NOT bLidSealerHommed;
	IF bLidSealerHommed THEN
		VIS.bLidSealerHeightSet:=TRUE;
		IF P06_LidSealer.fbLidSealer.eState=E_Station.eHomingDone AND P06_LidSealer.fbLidSealer2.eState=E_Station.eHomingDone THEN
			VIS.bLidSealerHeightSet:=FALSE;
			bLidSealerHommed:=FALSE;
			bLidSealerDoHoming:=FALSE;
			VIS.bLidSealerHoming:=FALSE;
		END_IF
	ELSIF P06_LidSealer.fbLidSealer.eState=E_Station.eHomingDone AND P06_LidSealer.fbLidSealer2.eState=E_Station.eHomingDone THEN
		bLidSealerDoHoming:=FALSE;
		bLidSealerHommed:=TRUE;
	END_IF
END_IF
IF VIS.bLidSealerDragingHoming THEN
	bLidSealerDragingStationEnable:=TRUE;
	bLidSealerDragingStationDoHoming:=NOT bLidSealerDragingHommed;
	IF bLidSealerDragingHommed THEN
		IF P06_LidSealer.fbLidSealerDragStation.eState=E_Station.eHomingDone THEN
			bLidSealerDragingHommed:=FALSE;
			bLidSealerDragingStationDoHoming:=FALSE;
			VIS.bLidSealerDragingHoming:=FALSE;
		END_IF
	ELSIF P06_LidSealer.fbLidSealerDragStation.eState=E_Station.eHomingDone THEN
		bLidSealerDragingHommed:=TRUE;
	END_IF
END_IF

(** Procedura bazowania podajnika opakowań**)
(****P07_ROPP*******)
IF VIS_ROPP.bROPPFeederHoming THEN
	bROPPFeederEnable						:=	TRUE; 
	VIS_ROPP.bROPPFeederRun					:=	FALSE;
	bROPPFeederDoHoming :=NOT bROPPFeederHommed;
	IF bROPPFeederHommed THEN
		VIS_ROPP.bROPPFeederHeightSet		:=	TRUE;
		IF P07_ROPP.fbROPPFeeder.eState=E_Station.eHomingDone THEN
			VIS_ROPP.bROPPFeederHeightSet	:=	FALSE;
			bROPPFeederHommed				:=	FALSE;
			bROPPFeederDoHoming				:=	FALSE;
			VIS_ROPP.bROPPFeederHoming		:=	FALSE;
		END_IF
	ELSIF P07_ROPP.fbROPPFeeder.eState=E_Station.eHomingDone THEN
		bROPPFeederDoHoming					:=	FALSE;
		bROPPFeederHommed					:=	TRUE;
	END_IF;
END_IF

IF VIS_ROPP.bROPPDragHoming THEN
	bROPPDragEnable							:=	TRUE; 
	VIS_ROPP.bROPPDragRun					:=	FALSE;
	bROPPDragDoHoming :=NOT bROPPDragHommed;
	IF bROPPDragHommed THEN
		IF P07_ROPP.fbROPPDrag.eState=E_Station.eHomingDone THEN
			bROPPDragHommed					:=	FALSE;
			bROPPDragDoHoming				:=	FALSE;
			VIS_ROPP.bROPPDragHoming		:=	FALSE;
		END_IF
	ELSIF P07_ROPP.fbROPPDrag.eState=E_Station.eHomingDone THEN
		bROPPDragHommed					:=	TRUE;
	END_IF;
END_IF

IF VIS_ROPP.bROPPCappingHoming THEN
	bROPPCappingEnable						:=	TRUE; 
	VIS_ROPP.bROPPCappingRun1				:=	FALSE;
	VIS_ROPP.bROPPCappingRun2				:=	FALSE;
	bROPPCappingDoHoming :=NOT bROPPCappingHommed;
	IF bROPPCappingHommed THEN
		VIS_ROPP.bROPPCappingHeightSet		:=	TRUE;
		IF P07_ROPP.fbROPPCapping.eState=E_Station.eHomingDone THEN
			VIS_ROPP.bROPPCappingHeightSet	:=	FALSE;
			bROPPCappingHommed				:=	FALSE;
			bROPPCappingDoHoming				:=	FALSE;
			VIS_ROPP.bROPPCappingHoming		:=	FALSE;
		END_IF
	ELSIF P07_ROPP.fbROPPCapping.eState=E_Station.eHomingDone THEN
		bROPPCappingDoHoming					:=	FALSE;
		bROPPCappingHommed					:=	TRUE;
	END_IF;
END_IF

(*****P08_CapFeeder********)
(******* Procedura bazowania stacji podajnika nakrętek ********)
IF VIS.bCapFeederHoming THEN
	bCapFeederEnable:=TRUE;
	bCapFeederDoHoming:=NOT bCapFeederHommed;
	IF bCapFeederHommed THEN
		VIS.bCapFeederHeightSet:=TRUE;
		IF P08_CapFeeder.fbCapFeeder.eState=E_Station.eHomingDone THEN
			VIS.bCapFeederHeightSet:=FALSE;
			bCapFeederHommed:=FALSE;
			bCapFeederDoHoming:=FALSE;
			VIS.bCapFeederHoming:=FALSE;
		END_IF
	ELSIF P08_CapFeeder.fbCapFeeder.eState=E_Station.eHomingDone THEN
			bCapFeederDoHoming:=FALSE;
			bCapFeederHommed:=TRUE;
	END_IF
END_IF

(*****P08_CapSorter********)
(******* Procedura bazowania stacji przeciagania pod sorterem nakrętek ********)
IF VIS.bCapSorterDragHoming THEN
	GVL.bCapSorterDragEnable:=TRUE; (*Włączenie enabla i kasowanie rozkazów*)
	VIS.bCapSorterDragRun:=FALSE;
	GVL.bCapSorterDragPrepareRun:=FALSE;
	bCapSorterDragDoHoming:=NOT bCapSorterDragHommed;
	IF bCapSorterDragHommed THEN
		IF P08_CapSorter.fbCapSorterDragStation.eState=E_Station.eHomingDone THEN
			VIS.bCapSorterDragHoming:=FALSE;
			bCapSorterDragHommed:=FALSE;
		END_IF
	ELSIF P08_CapSorter.fbCapSorterDragStation.eState=E_Station.eHomingDone THEN
			bCapSorterDragHommed:=TRUE;
	END_IF
END_IF

(******* Procedura bazowania stacji sortera nakrętek ********)
tonCapSorterHomingAndDone (IN:= stCapSorterWrite.bHoming, PT:=T#5S);
IF tonCapSorterHomingAndDone.Q THEN	
	IF stCapSorterRead.bHomingDone THEN
		stCapSorterWrite.bHoming 			:= FALSE;
	END_IF	
END_IF


(****************************************)
(***** 	P09_CapPuttedCheck	*******)
IF VIS.bCapPuttedCheckHoming THEN
	bCapPuttedCheckEnable:=TRUE; (*Włączenie enabla i kasowanie rozkazów*)
	bCapPuttedCheckDoHoming:=NOT bCapPuttedCheckHommed;
	IF bCapPuttedCheckHommed THEN
		VIS.bCapPuttedCheckHeightSet:=TRUE;
		IF P09_CapPuttedCheck.fbCapPuttedCheck.eState=E_Station.eHomingDone THEN
			VIS.bCapPuttedCheckHeightSet:=FALSE;
			bCapPuttedCheckHommed:=FALSE;
			bCapPuttedCheckDoHoming:=FALSE;
			VIS.bCapPuttedCheckHoming:=FALSE;
		END_IF
	ELSIF P09_CapPuttedCheck.fbCapPuttedCheck.eState=E_Station.eHomingDone THEN
			bCapPuttedCheckDoHoming:=FALSE;
			bCapPuttedCheckHommed:=TRUE;		
	END_IF
END_IF


(*****P10_GripperScrewers********)
(******* Procedura bazowania stacji przeciągania formatek z butelkami*******)
IF VIS.bBottleDragingStationHoming THEN
	GVL.bBottleDragingStationEnable:=TRUE; (*Włączenie enabla i kasowanie rozkazów*)
	VIS.bBottleDragingStationRun:=FALSE;
	GVL.bBottleDragingStationPrepareRun:=FALSE;
	bBottleDragingStationDoHoming:=NOT bBottleDragHommed;
	IF bBottleDragHommed THEN
		IF P10_GripperScrewer.fbGripperScrewersDragStation.eState=E_Station.eHomingDone (*AND P10_GripperScrewer.fbFormsDragingPneumaticStation.bHomingDone *)THEN
			bBottleDragHommed:=FALSE;
			bBottleDragingStationDoHoming:=FALSE;
			VIS.bBottleDragingStationHoming:=FALSE;
		END_IF
	ELSIF P10_GripperScrewer.fbGripperScrewersDragStation.eState=E_Station.eHomingDone  (*AND P10_GripperScrewer.fbFormsDragingPneumaticStation.bHomingDone*) THEN
		//	bBottleDragingStationDoHoming:=FALSE;
			bBottleDragHommed:=TRUE;
	END_IF
END_IF


(*****P10_GripperScrewers********)
(******* Procedura bazowania stacji zakecarki szczekowej*******)
IF VIS.bGripperScrewerHoming THEN
	VIS.bGripperScrewer1Run:=FALSE;
	VIS.bGripperScrewer2Run:=FALSE;
	bGripperScrewer1Enable:=TRUE;
	bGripperScrewer2Enable:=TRUE;
	bGripperScrewer1Catch:= FALSE;
	bGripperScrewer2Catch:=FALSE;
	bGripperScrewerDoHoming:=NOT bGripperScrewerHommed;
	IF bGripperScrewerHommed THEN
		VIS.bGripperScrewerCatchHeightSet:=TRUE;
		IF (P10_GripperScrewer.fbGripperScrewer1CatchStation.eState=E_Station.eHomingDone AND P10_GripperScrewer.fbGripperScrewer2CatchStation.eState=E_Station.eHomingDone) THEN
			VIS.bGripperScrewerHeightSet:=TRUE;
			IF P10_GripperScrewer.fb2GripperScrewer1.eState= E_Station.eHomingDone AND P10_GripperScrewer.fb2GripperScrewer2.eState= E_Station.eHomingDone THEN
				bGripperScrewerHommed:=FALSE;
				VIS.bGripperScrewerHeightSet:=FALSE;
				VIS.bGripperScrewerCatchHeightSet:=FALSE;
				bGripperScrewerDoHoming:=FALSE;
				VIS.bGripperScrewerHoming:=FALSE;
			END_IF
		END_IF
		//27.07.2022 dodałem warunek, że przy bazowaniu musi pojechać najpierw podnośnik na żądana wyskokość 
	ELSIF NOT bGripperScrewerHommed AND (P10_GripperScrewer.fb2GripperScrewer1.eState=E_Station.eHomingDone AND P10_GripperScrewer.fb2GripperScrewer2.eState=E_Station.eHomingDone) AND VIS.lrGripperScrewer1LiftActPos>=(P10_GripperScrewer.fb2GripperScrewer1.lrMaxHeightPosition-5)	AND VIS.lrGripperScrewer2LiftActPos>=(P10_GripperScrewer.fb2GripperScrewer2.lrMaxHeightPosition-5)	 THEN 
			bGripperScrewerCatch1DoHoming:=bGripperScrewerCatch2DoHoming:=TRUE;
		IF (P10_GripperScrewer.fbGripperScrewer1CatchStation.eState=E_Station.eHomingDone AND P10_GripperScrewer.fbGripperScrewer2CatchStation.eState=E_Station.eHomingDone)THEN
			//bGripperScrewerDoHoming:=FALSE;
			GVL.bGripperScrewerCatch1Homing:=GVL.bGripperScrewerCatch2Homing:=FALSE;
			bGripperScrewerCatch1DoHoming:=bGripperScrewerCatch2DoHoming:=FALSE;
			bGripperScrewerHommed:=TRUE;	
		END_IF	
	END_IF
END_IF
(****************************************)

(******	Procedura bazowania stacji	******)
(******	P11_CapCorrectCheck******)
IF VIS.bCapCorrectCheckHoming THEN
	bCapCorrectCheckEnable:=TRUE; (*Włączenie enabla i kasowanie rozkazów*)
	bCapCorrectCheckDoHoming:=NOT bCapCorrectCheckHommed;
	IF bCapCorrectCheckHommed THEN
		VIS.bCapCorrectCheckHeightSet:=TRUE;
		IF P11_CapCorrectCheck.fbCapCorrectCheck.eState=E_Station.eHomingDone THEN
			VIS.bCapCorrectCheckHeightSet:=FALSE;
			bCapCorrectCheckHommed:=FALSE;
			bCapCorrectCheckDoHoming:=FALSE;
			VIS.bCapCorrectCheckHoming:=FALSE;
		END_IF
	ELSIF P11_CapCorrectCheck.fbCapCorrectCheck.eState=E_Station.eHomingDone THEN
			bCapCorrectCheckDoHoming:=FALSE;
			bCapCorrectCheckHommed:=TRUE;		
	END_IF
END_IF
(****************************************)


(******	Procedura bazowania stacji	******)
(******	P13_BottleTransfer******)
IF VIS.bBottleTransferHoming THEN
	bBottleTransferEnable:=TRUE;
	VIS.bBottleTransferPlace:=FALSE;	
	VIS.bBottleTransferRun:=FALSE;	
	bBottleTransferDoHoming:=NOT bBottleTransferHommed;
	IF bBottleTransferHommed THEN
		VIS.bBottleTransferHeightSet:=TRUE;
		IF P13_BottleTransfer.fbBottleTransfer.eState=E_Station.eHomingDone THEN
			VIS.bBottleTransferHeightSet:=FALSE;
			bBottleTransferHommed:=FALSE;
			bBottleTransferDoHoming:=FALSE;
			VIS.bBottleTransferHoming:=FALSE;
		END_IF
	ELSIF P13_BottleTransfer.fbBottleTransfer.eState=E_Station.eHomingDone THEN
			bBottleTransferDoHoming:=FALSE;
			bBottleTransferHommed :=TRUE;		
			VIS.bBottleTransferHoming:=FALSE;
	END_IF
END_IF
(****************************************)
END_ACTION

ACTION ACT_ResetAfterError:

 (*Zachowanie po stopie awaryjnym*)
IF P00_Alarms.arfbAlarm[1].bActive THEN
	iGripperScrewerCase := 0; // Bo za szybko zaczeło chwytać
END_IF

 (*Zachowanie po stopie awaryjnym*)
 IF P00_Alarms.arfbAlarm[1].bActive THEN
     //Jezeli było w trakcie dozowania i coś wydozowało
     IF (iDispencersCase = 4 ) OR (lrDosedMass1CVAux>2 OR lrDosedMass2CVAux>2 OR lrDosedMass3CVAux>2 OR lrDosedMass4CVAux > 2) THEN
         eDispencersPackageState[4].bDoseAborted:=TRUE;
         eDispencersPackageState[3].bDoseAborted:=TRUE;
         eDispencersPackageState[2].bDoseAborted:=TRUE;
         eDispencersPackageState[1].bDoseAborted:=TRUE;
     END_IF
 END_IF
 (*Zachowanie po jakimkolwiek błędzie dozownika 1 i dozownika 2*)
 IF P00_Alarms.aLastStationsErrors[9].bError OR P00_Alarms.aLastStationsErrors[10].bError OR P00_Alarms.aLastStationsErrors[11].bError OR P00_Alarms.aLastStationsErrors[12].bError  THEN
     //Jezeli było w trakcie dozowania i coś wydozowało
     IF (iDispencersCase = 4 ) OR (ABS(lrDosedMass1CVAux)>2 OR ABS(lrDosedMass2CVAux)>2 OR ABS(lrDosedMass3CVAux)>2 OR ABS(lrDosedMass4CVAux) > 2) THEN
         eDispencersPackageState[4].bDoseAborted:=TRUE;
         eDispencersPackageState[3].bDoseAborted:=TRUE;
         eDispencersPackageState[2].bDoseAborted:=TRUE;
         eDispencersPackageState[1].bDoseAborted:=TRUE;
     END_IF
 END_IF
  (*Zachowanie po błędzie przeciagania*)
 IF P00_Alarms.aLastStationsErrors[4].bError OR P00_Alarms.aLastStationsErrors[41].bError OR P00_Alarms.arfbAlarm[41].bActive THEN //Prawe/Lewe
         eBeforeDispencersPackageState[4].bDoseAborted:=TRUE;
         eBeforeDispencersPackageState[3].bDoseAborted:=TRUE;
         eBeforeDispencersPackageState[2].bDoseAborted:=TRUE;
         eBeforeDispencersPackageState[1].bDoseAborted:=TRUE;
     	 eDispencersPackageState[4].bDoseAborted:=TRUE;
         eDispencersPackageState[3].bDoseAborted:=TRUE;
         eDispencersPackageState[2].bDoseAborted:=TRUE;
         eDispencersPackageState[1].bDoseAborted:=TRUE;		  
 END_IF
 
(*Zachowanie po błędzie sortera nasadek*)
 IF P00_Alarms.aLastStationsErrors[50].bError THEN
	
		iCapSorterCase := 0;
		eCapSorterPackageState[1].bCapSorterPuttedAborted	:=	TRUE;
		eCapSorterPackageState[2].bCapSorterPuttedAborted	:=	TRUE;
		eCapSorterPackageState[3].bCapSorterPuttedAborted	:=	TRUE;
		eCapSorterPackageState[4].bCapSorterPuttedAborted	:=	TRUE;
	
 END_IF
 
 (*Zachowanie po błędzie przeciągania sortera nasadek*)	(*Błąd zablokowanej nasadki*)
 IF P00_Alarms.aLastStationsErrors[51].bError OR P00_Alarms.arfbAlarm[35].bActive THEN
	
		eCapSorterPackageState[1].bCapSorterPuttedAborted	:=	TRUE;
		eCapSorterPackageState[2].bCapSorterPuttedAborted	:=	TRUE;
		eCapSorterPackageState[3].bCapSorterPuttedAborted	:=	TRUE;
		eCapSorterPackageState[4].bCapSorterPuttedAborted	:=	TRUE;

		eBeforeCapSorterPackageState[1].bCapSorterPuttedAborted	:=	TRUE;
		eBeforeCapSorterPackageState[2].bCapSorterPuttedAborted	:=	TRUE;
		eBeforeCapSorterPackageState[3].bCapSorterPuttedAborted	:=	TRUE;
		eBeforeCapSorterPackageState[4].bCapSorterPuttedAborted	:=	TRUE;
		
 END_IF
END_ACTION

ACTION ACT_ResetAfterErrorOrEstop_do_usun:

 (*Zachowanie po stopie awaryjnym*)
IF P00_Alarms.aLastStationsErrors[1].nErrorCode = 1 THEN
	iGripperScrewerCase := 0; // Bo za szybko zaczeło chwytać
END_IF

 (*Zachowanie po stopie awaryjnym*)
 IF P00_Alarms.aLastStationsErrors[1].nErrorCode >= 1 AND P00_Alarms.aLastStationsErrors[1].nErrorCode <= 20 THEN
     //Jezeli było w trakcie dozowania i coś wydozowało
     IF (iDispencersCase = 4 ) OR (lrDosedMass1CVAux>2 OR lrDosedMass2CVAux>2 OR lrDosedMass3CVAux>2 OR lrDosedMass4CVAux > 2) THEN
         eDispencersPackageState[4].bDoseAborted:=TRUE;
         eDispencersPackageState[3].bDoseAborted:=TRUE;
         eDispencersPackageState[2].bDoseAborted:=TRUE;
         eDispencersPackageState[1].bDoseAborted:=TRUE;
     END_IF
 END_IF
 (*Zachowanie po jakimkolwiek błędzie dozownika 1 i dozownika 2*)
 IF P00_Alarms.aLastStationsErrors[9].bError OR P00_Alarms.aLastStationsErrors[10].bError OR P00_Alarms.aLastStationsErrors[11].bError OR P00_Alarms.aLastStationsErrors[12].bError  THEN
     //Jezeli było w trakcie dozowania i coś wydozowało
     IF (iDispencersCase = 4 ) OR (ABS(lrDosedMass1CVAux)>2 OR ABS(lrDosedMass2CVAux)>2 OR ABS(lrDosedMass3CVAux)>2 OR ABS(lrDosedMass4CVAux) > 2) THEN
         eDispencersPackageState[4].bDoseAborted:=TRUE;
         eDispencersPackageState[3].bDoseAborted:=TRUE;
         eDispencersPackageState[2].bDoseAborted:=TRUE;
         eDispencersPackageState[1].bDoseAborted:=TRUE;
     END_IF
 END_IF
  (*Zachowanie po błędzie przeciagania*)
 IF P00_Alarms.aLastStationsErrors[4].bError OR P00_Alarms.aLastStationsErrors[41].bError OR (P00_Alarms.aLastStationsErrors[1].bError AND P00_Alarms.aLastStationsErrors[1].nErrorCode=70)THEN //Prawe/Lewe
         eBeforeDispencersPackageState[4].bDoseAborted:=TRUE;
         eBeforeDispencersPackageState[3].bDoseAborted:=TRUE;
         eBeforeDispencersPackageState[2].bDoseAborted:=TRUE;
         eBeforeDispencersPackageState[1].bDoseAborted:=TRUE;
     	 eDispencersPackageState[4].bDoseAborted:=TRUE;
         eDispencersPackageState[3].bDoseAborted:=TRUE;
         eDispencersPackageState[2].bDoseAborted:=TRUE;
         eDispencersPackageState[1].bDoseAborted:=TRUE;		  
 END_IF
 
(*Zachowanie po błędzie sortera nasadek*)
 IF P00_Alarms.aLastStationsErrors[50].bError THEN
	
		iCapSorterCase := 0;
		eCapSorterPackageState[1].bCapSorterPuttedAborted	:=	TRUE;
		eCapSorterPackageState[2].bCapSorterPuttedAborted	:=	TRUE;
		eCapSorterPackageState[3].bCapSorterPuttedAborted	:=	TRUE;
		eCapSorterPackageState[4].bCapSorterPuttedAborted	:=	TRUE;
	
 END_IF
 
 (*
 (*Zachowanie po błędzie przeciągania sortera nasadek*)	(*Błąd zablokowanej nasadki*)
 IF P00_Alarms.aLastStationsErrors[51].bError OR (P00_Alarms.aLastStationsErrors[1].bError AND P00_Alarms.aLastStationsErrors[1].nErrorCode=64) THEN
	
		eCapSorterPackageState[1].bCapSorterPuttedAborted	:=	TRUE;
		eCapSorterPackageState[2].bCapSorterPuttedAborted	:=	TRUE;
		eCapSorterPackageState[3].bCapSorterPuttedAborted	:=	TRUE;
		eCapSorterPackageState[4].bCapSorterPuttedAborted	:=	TRUE;

		eBeforeCapSorterPackageState[1].bCapSorterPuttedAborted	:=	TRUE;
		eBeforeCapSorterPackageState[2].bCapSorterPuttedAborted	:=	TRUE;
		eBeforeCapSorterPackageState[3].bCapSorterPuttedAborted	:=	TRUE;
		eBeforeCapSorterPackageState[4].bCapSorterPuttedAborted	:=	TRUE;
	
 END_IF
 *)
END_ACTION

ACTION ACT_ResetAfterStart:
	IF rtResetAfterStart.Q THEN //po 60s
		
		GVL.eCapSorterPackageState[1] 				:= GVL.eClearPackageState;
		GVL.eCapSorterPackageState[2] 				:= GVL.eClearPackageState;
		GVL.eCapSorterPackageState[3] 				:= GVL.eClearPackageState;
		GVL.eCapSorterPackageState[4] 				:= GVL.eClearPackageState;	
	
		GVL.eBeforeCapSorterPackageState[1] 		:= GVL.eClearPackageState;
		GVL.eBeforeCapSorterPackageState[2] 		:= GVL.eClearPackageState;
		GVL.eBeforeCapSorterPackageState[3] 		:= GVL.eClearPackageState;
		GVL.eBeforeCapSorterPackageState[4] 		:= GVL.eClearPackageState;
	
		GVL.eWeightPackageState[1] 					:= GVL.eClearPackageState;
		GVL.eWeightPackageState[2] 					:= GVL.eClearPackageState;
		GVL.eWeightPackageState[3] 					:= GVL.eClearPackageState;
		GVL.eWeightPackageState[4] 					:= GVL.eClearPackageState;

		GVL.eAfterDispencersPackageState[1]			:= GVL.eClearPackageState;
		GVL.eAfterDispencersPackageState[2]			:= GVL.eClearPackageState;
		GVL.eAfterDispencersPackageState[3]			:= GVL.eClearPackageState;	
		GVL.eAfterDispencersPackageState[4]			:= GVL.eClearPackageState;	
	
	
		eBeforeLidFeeder2PackageState[4]			:= GVL.eClearPackageState;		
		eBeforeLidFeeder2PackageState[3]			:= GVL.eClearPackageState;	
		eBeforeLidFeeder2PackageState[2]			:= GVL.eClearPackageState;	
		eBeforeLidFeeder2PackageState[1]			:= GVL.eClearPackageState;	
			
		eBeforeLidFeederPackageState[2]				:= GVL.eClearPackageState;		
		eBeforeLidFeederPackageState[1]				:= GVL.eClearPackageState;		
				
		eLidFeederPackageState[2]					:= GVL.eClearPackageState;		
		eLidFeederPackageState[1]					:= GVL.eClearPackageState;		
				
		eAfterLidFeederPackageState[2]				:= GVL.eClearPackageState;	
		eAfterLidFeederPackageState[1]				:= GVL.eClearPackageState;		
				
		eBeforeLidSealerPackageState[2]				:= GVL.eClearPackageState;		
		eBeforeLidSealerPackageState[1]				:= GVL.eClearPackageState;		
				
		eLidSealerPackageState[2]					:= GVL.eClearPackageState;	
		eLidSealerPackageState[1]					:= GVL.eClearPackageState;	
		
		(*Ustawianie licznika zależnie od czujnika*)
		//IF fbIbCapPuttedCheckFormSensor.bOUT THEN	//Czujnik 5 formatki przed zakrecarkami 
		//	VIS.iNumbersOfFormsBetweenWeightAndScrewers := 1;
		//ELSE
			VIS.iNumbersOfFormsBetweenWeightAndScrewers := 0;
		//END_IF
		irtResetAfterStart	:=	irtResetAfterStart	+	1;
	END_IF
END_ACTION

ACTION ACT_ResetCommands:
(*Resetowanie wszystkich rozkazów*)
(*Zachować kolejność stacji*)



ACT_ResetCommandsHoming();

//Czy na pewno kasowac?
//VIS.bMachinePartsChangeover				:=FALSE;

VIS.bAllowStart:=FALSE;
VIS.bCheckStart:=FALSE;
VIS.bRecipeLoading:=FALSE;

VIS.bCapSorterEmptyingMode				:= FALSE;		
VIS.bBottleSorterEmptyingMode			:= FALSE;	
bCapSorterBottleSorterAutoStart			:= FALSE;
P06_LidSealer.bMovetoEndPositionLidSealer	:=FALSE;
P06_LidFeeder.bMovetoEndPositionLidFeeder	:=FALSE;
(********** Pack_ML*************)
//iStoppingCase							:= 0;
bDelayAfterStart						:= FALSE;
iWeightCase								:= 0;
brtLongDelayFirstDraging				:= FALSE;
bFirstDragingWickFeederAfterRestart1	:= FALSE;
bFirstDragingLidFeederAfterRestart1		:= FALSE;
bFirstDragingLidFeederAfterRestart2		:= FALSE;
bFirstDragingLidSealerAfterRestart1		:= FALSE;
bFirstDragingLidSealerAfterRestart2		:= FALSE;
iFirstDragingLidFeederAfterRestart2Count:=0;
iFirstDragingLidSealerAfterRestart2Count:=0;

